Omron CX-Programmer project 新工程 (CX-Programmer 9.42)

# PLC 新PLC1: CP1E N60

## Global symbols (name address type ; comment)
0.04 BOOL  ; 0轴DO2备用
0.06 BOOL  ; 0轴Z相输出
0.07 BOOL  ; 1轴Z相输出
0.10 BOOL  ; 0轴接近零位开关
0.11 BOOL  ; 1轴接近零位开关
100.00 BOOL  ; 0轴脉冲指令
100.01 BOOL  ; 1轴脉冲指令
100.02 BOOL  ; 0轴脉冲方向
100.03 BOOL  ; 1轴脉冲方向
1.04 BOOL  ; 1轴DO2备用
4.10 BOOL  ; 备用
A276 CHANNEL  ; 脉冲输出0的当前值(PV)
A277 CHANNEL  ; 脉冲输出0的当前值(PV)
A278 CHANNEL  ; 脉冲输出1的当前值(PV)
A279 CHANNEL  ; 脉冲输出1的当前值(PV)
A280.00 BOOL  ; 脉冲输出0加速/减速标志
A280.01 BOOL  ; 脉冲输出0上溢/下溢标志
A280.02 BOOL  ; 脉冲输出0输出量设定标志
A280.03 BOOL  ; 脉冲输出0输出完成标志
A280.04 BOOL  ; 脉冲输出0输出中标志
A280.05 BOOL  ; 脉冲输出0无原点标志
A280.06 BOOL  ; 脉冲输出0停止在原点标志
A280.07 BOOL  ; 脉冲输出0输出停止出错标志
A281.00 BOOL  ; 脉冲输出1加速/减速标志
A281.01 BOOL  ; 脉冲输出1上溢/下溢标志
A281.03 BOOL  ; 脉冲输出1输出完成标志
A281.04 BOOL  ; 脉冲输出1输出中标志
A281.05 BOOL  ; 脉冲输出1无原点标志
A281.06 BOOL  ; 脉冲输出1停止在原点标志
A281.07 BOOL  ; 脉冲输出1输出停止出错标志
A444 CHANNEL  ; 脉冲输出0停止出错代码
A445 CHANNEL  ; 脉冲输出1停止出错代码
A540.00 BOOL  ; 脉冲输出0复位位
A540.08 BOOL  ; 脉冲输出0CW限位输入信号标志
A540.09 BOOL  ; 脉冲输出0CCW限位输入信号标志
A540.10 BOOL  ; 脉冲输出0定位完成信号
A541.00 BOOL  ; 脉冲输出1复位位
A541.08 BOOL  ; 脉冲输出1CW限位输入信号标志
A541.09 BOOL  ; 脉冲输出1CCW限位输入信号标志
A541.10 BOOL  ; 脉冲输出1定位完成信号
T201 BOOL  ; 阻挡片气缸1电磁阀
T202 BOOL  ; 阻挡片气缸2电磁阀
T203 BOOL  ; 阻挡片气缸3电磁阀
T204 BOOL  ; 盒子顶出气缸电磁阀
T205 BOOL  ; 机器手气缸1电磁阀
T206 BOOL  ; 机器手气缸2电磁阀
T207 BOOL  ; 旋转90度阻挡气缸1电磁阀
T208 BOOL  ; 旋转90度阻挡气缸2电磁阀
T209 BOOL  ; 上料真空电磁阀
T210 BOOL  ; 下料真空电磁阀
T211 BOOL  ; 吹气电磁阀
T220 BOOL  ; 盒子顶出气缸电磁阀顶出延时
T221 BOOL  ; 盒子顶出气缸电磁阀退回延时
T222 BOOL  ; 光纤物品检测感应2通过延时
T223 BOOL  ; 光纤物品检测感应2顶升延时1
T224 BOOL  ; 机械手1顶出延时1
T225 BOOL  ; 机械手1退回延时1
T226 BOOL  ; 光纤物品检测感应2顶升延时2
T227 BOOL  ; 光纤物品检测感应2顶升延时3
T228 BOOL  ; 开始延时
T229 BOOL  ; 机械手1延时1
T230 BOOL  ; 机械手1延时2
T231 BOOL  ; 机械手1延时3
T232 BOOL  ; 机械手1延时4
T233 BOOL  ; 机械手1延时5
T234 BOOL  ; 机械手1顶出延时2
T235 BOOL  ; 机械手1退回延时2
T236 BOOL  ; 机械手2顶出延时1
T237 BOOL  ; 机械手2退回延时1
T238 BOOL  ; 机械手2顶出延时2
T239 BOOL  ; 机械手2退回延时2
T240 BOOL  ; 机械手2顶出延时3
T241 BOOL  ; 机械手2退回延时3
T242 BOOL  ; 机械手2顶出延时4
T243 BOOL  ; 机械手2退回延时4
T244 BOOL  ; 机械手2顶出延时5
T245 BOOL  ; 机械手2退回延时5
T246 BOOL  ; 机械手2顶出延时6
T247 BOOL  ; 机械手2退回延时6
B_0_ACC_CCW_run 29.05 BOOL  ; 0轴反向运行
B_0_ACC_CW_run 29.03 BOOL  ; 0轴正向运行
B_0_CCW_Interlock 29.08 BOOL  ; 0轴CCW互锁
B_0_CCW_manual 29.14 BOOL  ; 0轴反向手动点动
B_0_CCW_manualing 30.02 BOOL  ; 0轴反向手动点动中
B_0_CW_Interlock 29.07 BOOL  ; 0轴CW互锁
B_0_CW_manual 29.13 BOOL  ; 0轴正向手动点动
B_0_CW_manualing 30.01 BOOL  ; 0轴正向手动点动中
B_0_ORG_POS 31.04 BOOL  ; 0轴原点位置
B_0_ORG_search 30.05 BOOL  ; 0轴原点搜索
B_0_ORG_searched 30.07 BOOL  ; 0轴原点搜索完成
B_0_ORG_searching 30.06 BOOL  ; 0轴原点搜索中
B_0_ORG_seted 30.08 BOOL  ; 0轴原点已定义
B_0_PLS2_CCW_run 28.13 BOOL  ; 0轴反向运行
B_0_PLS2_CW_run 28.11 BOOL  ; 0轴正向运行
B_0_SPED_CCW_run 29.01 BOOL  ; 0轴反向运行
B_0_SPED_CW_run 28.15 BOOL  ; 0轴正向运行
B_0_SRV_ON 31.00 BOOL  ; 0轴伺服ON
B_0_drive_stop 29.11 BOOL  ; 0轴运行停止
B_1_ACC_CCW_run 29.06 BOOL  ; 1轴反向运行
B_1_ACC_CW_run 29.04 BOOL  ; 1轴正向运行
B_1_CCW_Interlock 29.10 BOOL  ; 1轴CCW互锁
B_1_CCW_manual 30.00 BOOL  ; 1轴反向手动点动
B_1_CCW_manualing 30.04 BOOL  ; 1轴反向手动点动中
B_1_CW_Interlock 29.09 BOOL  ; 1轴CW互锁
B_1_CW_manual 29.15 BOOL  ; 1轴正向手动点动
B_1_CW_manualing 30.03 BOOL  ; 1轴正向手动点动中
B_1_ORG_POS 31.05 BOOL  ; 1轴原点位置
B_1_ORG_search 30.09 BOOL  ; 1轴原点搜索
B_1_ORG_searched 30.11 BOOL  ; 1轴原点搜索完成
B_1_ORG_searching 30.10 BOOL  ; 1轴原点搜索中
B_1_ORG_seted 30.12 BOOL  ; 1轴原点已定义
B_1_PLS2_CCW_run 28.14 BOOL  ; 1轴反向运行
B_1_PLS2_CW_run 28.12 BOOL  ; 1轴正向运行
B_1_SPED_CCW_run 29.02 BOOL  ; 1轴反向运行
B_1_SPED_CW_run 29.00 BOOL  ; 1轴正向运行
B_1_SRV_ON 31.01 BOOL  ; 1轴伺服ON
B_1_drive_stop 29.12 BOOL  ; 1轴运行停止
B_LL_1 43.11 BOOL  ; 落料位1
B_LL_2 43.12 BOOL  ; 落料位2
B_LL_3 43.13 BOOL  ; 落料位3
B_LL_4 43.14 BOOL  ; 落料位4
B_POS_DONE 31.03 BOOL  ; 定位结束
B_POS_START_INS 31.02 BOOL  ; 定位开始指令
B_SRV_enabled 30.14 BOOL  ; 伺服自动使能
B_SRV_reset 30.15 BOOL  ; 伺服控制复位
B_SYS_24V_ERR_1 21.04 BOOL  ; 系统24V故障区域1
B_SYS_24V_ERR_2 21.05 BOOL  ; 系统24V故障区域2
B_SYS_24V_ERR_3 21.06 BOOL  ; 系统24V故障区域3
B_SYS_ON_ERR 21.01 BOOL  ; 系统开机故障
B_SYS_RD 20.08 BOOL  ; 系统就绪
B_SYS_airbreaker 20.09 BOOL  ; 系统断路器正常（总）
B_SYS_auto 20.07 BOOL  ; 系统自动（总）
B_SYS_door_ask 20.10 BOOL  ; 系统维修门开门请求（总）
B_SYS_emergency 20.11 BOOL  ; 系统急停（总）
B_SYS_erroring 21.03 BOOL  ; 系统故障中（总）
B_SYS_hold 20.05 BOOL  ; 系统暂停（总）
B_SYS_home 20.12 BOOL  ; 系统工作原点（总）
B_SYS_manual 20.06 BOOL  ; 系统手动（总）
B_SYS_off 20.13 BOOL  ; 系统关机
B_SYS_on 20.14 BOOL  ; 系统开机
B_SYS_oning 20.15 BOOL  ; 系统开机中
B_SYS_reset 20.04 BOOL  ; 系统复位（总）
B_SYS_running 21.00 BOOL  ; 系统运行中
B_SYS_single_cycle 28.10 BOOL  ; 系统单循环（总）
B_SYS_start 20.02 BOOL  ; 系统启动（总）
B_SYS_start_ERR 21.02 BOOL  ; 系统开始故障
B_SYS_stop 20.03 BOOL  ; 系统停止（总）
B_SYS_stoping 20.00 BOOL  ; 系统停止中
B_jog_enabled 30.13 BOOL  ; 手动点动使能
D_0_CCW_acc_Freq 32 DWORD  ; 0轴反向acc目标频率
D_0_CCW_pls2_Freq D1122 DWORD  ; 0轴反向pls2目标频率
D_0_CCW_pls2_PUL D1124 DWORD  ; 0轴反向pls2输出脉冲
D_0_CCW_sped_Freq 38 UDINT  ; 0轴反向点动频率
D_0_CW_acc_Freq 40 DWORD  ; 0轴正向acc目标频率
D_0_CW_pls2_Freq D1102 DWORD  ; 0轴正向pls2目标频率
D_0_CW_pls2_PUL D1104 DWORD  ; 0轴正向pls2输出脉冲
D_0_CW_sped_Freq 46 UDINT  ; 0轴正向点动频率
D_0_user_point_Freq_00 D1000 DWORD  ; 0轴通用位置点频率00
D_0_user_point_Freq_01 D1004 DWORD  ; 0轴通用位置点频率01
D_0_user_point_Freq_02 D1008 DWORD  ; 0轴通用位置点频率02
D_0_user_point_Freq_03 D1012 DWORD  ; 0轴通用位置点频率03
D_0_user_point_Freq_04 D1016 DWORD  ; 0轴通用位置点频率04
D_0_user_point_Freq_05 D1020 DWORD  ; 0轴通用位置点频率05
D_0_user_point_PUL_00 D1002 DWORD  ; 0轴通用位置点脉冲00
D_0_user_point_PUL_01 D1006 DWORD  ; 0轴通用位置点脉冲01
D_0_user_point_PUL_02 D1010 DWORD  ; 0轴通用位置点脉冲02
D_0_user_point_PUL_03 D1014 DWORD  ; 0轴通用位置点脉冲03
D_0_user_point_PUL_04 D1018 DWORD  ; 0轴通用位置点脉冲04
D_0_user_point_PUL_05 D1022 DWORD  ; 0轴通用位置点脉冲05
D_1_CCW_acc_Freq 52 DWORD  ; 1轴反向acc目标频率
D_1_CCW_pls2_Freq D1128 DWORD  ; 1轴反向pls2目标频率
D_1_CCW_pls2_PUL D1130 DWORD  ; 1轴反向pls2输出脉冲
D_1_CCW_sped_Freq 58 UDINT  ; 1轴反向点动频率
D_1_CW_acc_Freq 60 DWORD  ; 1轴正向acc目标频率
D_1_CW_pls2_Freq D1108 DWORD  ; 1轴正向pls2目标频率
D_1_CW_pls2_PUL D1110 DWORD  ; 1轴正向pls2输出脉冲
D_1_CW_sped_Freq 66 UDINT  ; 1轴正向点动频率
D_1_user_point_Freq_00 D1024 DWORD  ; 1轴通用位置点频率00
D_1_user_point_Freq_01 D1028 DWORD  ; 1轴通用位置点频率01
D_1_user_point_Freq_02 D1032 DWORD  ; 1轴通用位置点频率02
D_1_user_point_Freq_03 D1036 DWORD  ; 1轴通用位置点频率03
D_1_user_point_Freq_04 D1040 DWORD  ; 1轴通用位置点频率04
D_1_user_point_Freq_05 D1044 DWORD  ; 1轴通用位置点频率05
D_1_user_point_PUL_00 D1026 DWORD  ; 1轴通用位置点脉冲00
D_1_user_point_PUL_01 D1030 DWORD  ; 1轴通用位置点脉冲01
D_1_user_point_PUL_02 D1034 DWORD  ; 1轴通用位置点脉冲02
D_1_user_point_PUL_03 D1038 DWORD  ; 1轴通用位置点脉冲03
D_1_user_point_PUL_04 D1042 DWORD  ; 1轴通用位置点脉冲04
D_1_user_point_PUL_05 D1046 DWORD  ; 1轴通用位置点脉冲05
END_001_step 22.04 BOOL  ; 结束步01
END_002_step 22.05 BOOL  ; 结束步02
END_FIN_step 22.06 BOOL  ; 结束完成步
HMI_B_0_CCW_manual 132.13 BOOL  ; 0轴反向手动点动
HMI_B_0_CW_manual 132.12 BOOL  ; 0轴正向手动点动
HMI_B_0_ORG_search 132.03 BOOL  ; 0轴原点搜索
HMI_B_0_ORG_seted 132.04 BOOL  ; 0轴原点已定义
HMI_B_0_POS_set 133.02 BOOL  ; 0轴动作点设置
HMI_B_0_PWR_Oning 131.14 BOOL  ; 0轴已上电
HMI_B_0_SRV_ON 132.01 BOOL  ; 0轴伺服ON
HMI_B_0_SRV_Oning 132.00 BOOL  ; 0轴已伺服ON
HMI_B_0_alarm 131.15 BOOL  ; 0轴伺服报警
HMI_B_0_alarm_CLR 132.02 BOOL  ; 0轴警报清除
HMI_B_1_CCW_manual 132.15 BOOL  ; 1轴反向手动点动
HMI_B_1_CW_manual 132.14 BOOL  ; 1轴正向手动点动
HMI_B_1_ORG_search 132.10 BOOL  ; 1轴原点搜索
HMI_B_1_ORG_seted 132.11 BOOL  ; 1轴原点已定义
HMI_B_1_POS_set 133.03 BOOL  ; 1轴动作点设置
HMI_B_1_PWR_Oning 132.05 BOOL  ; 1轴已上电
HMI_B_1_SRV_ON 132.08 BOOL  ; 1轴伺服ON
HMI_B_1_SRV_Oning 132.07 BOOL  ; 1轴已伺服ON
HMI_B_1_alarm 132.06 BOOL  ; 1轴伺服报警
HMI_B_1_alarm_CLR 132.09 BOOL  ; 1轴警报清除
HMI_B_BJ1_QD 130.11 BOOL  ; 步进1启动
HMI_B_BJ1_YG 133.01 BOOL  ; 步进1用光
HMI_B_BJ1_ZQD 133.00 BOOL  ; 步进1再启动
HMI_B_BJ2_QD 130.12 BOOL  ; 步进2启动
HMI_B_BJ3_1 131.00 BOOL  ; 步进3计数器加1
HMI_B_BJ3_1_DONE 131.01 BOOL  ; 步进3计数器结束
HMI_B_BJ3_QD 130.13 BOOL  ; 步进3启动
HMI_B_BJ4_QD 130.14 BOOL  ; 步进4启动
HMI_B_CQF 130.10 BOOL  ; 吹气电磁阀
HMI_B_CQF_ALM 131.13 BOOL  ; 吹气电磁阀报警
HMI_B_DCQGF 130.03 BOOL  ; 盒子顶出气缸电磁阀
HMI_B_DCQGF_ALM 131.06 BOOL  ; 盒子顶出气缸电磁阀报警
HMI_B_PLC_DEBUG 131.02 BOOL  ; PLC单独调试
HMI_B_RBQGF1 130.04 BOOL  ; 机器手气缸1电磁阀
HMI_B_RBQGF1_ALM 131.07 BOOL  ; 机器手气缸1电磁阀报警
HMI_B_RBQGF2 130.05 BOOL  ; 机器手气缸2电磁阀
HMI_B_RBQGF2_ALM 131.08 BOOL  ; 机器手气缸2电磁阀报警
HMI_B_RD_TBC_BT 120.07 BOOL  ; HMI就绪确认
HMI_B_SYS_24V_ERR_1 121.12 BOOL  ; HMI系统24V故障区域1
HMI_B_SYS_24V_ERR_2 121.13 BOOL  ; HMI系统24V故障区域2
HMI_B_SYS_24V_ERR_3 121.14 BOOL  ; HMI系统24V故障区域3
HMI_B_SYS_ON_ERR 121.09 BOOL  ; HMI系统开机故障
HMI_B_SYS_RD 120.15 BOOL  ; HMI系统就绪
HMI_B_SYS_airbreaker 121.01 BOOL  ; HMI系统断路器正常（总）
HMI_B_SYS_auto 120.14 BOOL  ; HMI系统自动（总）
HMI_B_SYS_door_ask 121.02 BOOL  ; HMI系统维修门开门请求（总）
HMI_B_SYS_emergency 121.03 BOOL  ; HMI系统急停（总）
HMI_B_SYS_erroring 121.11 BOOL  ; HMI系统故障中（总）
HMI_B_SYS_hold 120.12 BOOL  ; HMI系统暂停（总）
HMI_B_SYS_home 121.04 BOOL  ; HMI系统工作原点（总）
HMI_B_SYS_manual 120.13 BOOL  ; HMI系统手动（总）
HMI_B_SYS_off 121.05 BOOL  ; HMI系统关机
HMI_B_SYS_on 121.06 BOOL  ; HMI系统开机
HMI_B_SYS_oning 121.07 BOOL  ; HMI系统开机中
HMI_B_SYS_reset 120.11 BOOL  ; HMI系统复位（总）
HMI_B_SYS_running 121.08 BOOL  ; HMI系统运行中
HMI_B_SYS_single_cycle 121.00 BOOL  ; HMI系统单循环（总）
HMI_B_SYS_start 120.09 BOOL  ; HMI系统启动（总）
HMI_B_SYS_start_ERR 121.10 BOOL  ; HMI系统开始故障
HMI_B_SYS_stop 120.10 BOOL  ; HMI系统停止（总）
HMI_B_XZQGF1 130.06 BOOL  ; 旋转90度阻挡气缸1电磁阀
HMI_B_XZQGF1_ALM 131.09 BOOL  ; 旋转90度阻挡气缸1电磁阀报警
HMI_B_XZQGF2 130.07 BOOL  ; 旋转90度阻挡气缸2电磁阀
HMI_B_XZQGF2_ALM 131.10 BOOL  ; 旋转90度阻挡气缸2电磁阀报警
HMI_B_ZDQGF1 130.00 BOOL  ; 阻挡片气缸1电磁阀
HMI_B_ZDQGF1_ALM 131.03 BOOL  ; 阻挡片气缸1电磁阀报警
HMI_B_ZDQGF2 130.01 BOOL  ; 阻挡片气缸2电磁阀
HMI_B_ZDQGF2_ALM 131.04 BOOL  ; 阻挡片气缸2电磁阀报警
HMI_B_ZDQGF3 130.02 BOOL  ; 阻挡片气缸3电磁阀
HMI_B_ZDQGF3_ALM 131.05 BOOL  ; 阻挡片气缸3电磁阀报警
HMI_B_ZKXP1 130.08 BOOL  ; 上料真空电磁阀
HMI_B_ZKXP1_ALM 131.11 BOOL  ; 上料真空电磁阀报警
HMI_B_ZKXP2 130.09 BOOL  ; 下料真空电磁阀
HMI_B_ZKXP2_ALM 131.12 BOOL  ; 下料真空电磁阀报警
HMI_B_auto_BT 120.05 BOOL  ; HMI自动按钮
HMI_B_belt_motor 130.15 BOOL  ; 皮带电机
HMI_B_emergency_BT 120.06 BOOL  ; HMI急停按钮
HMI_B_hold_BT 120.03 BOOL  ; HMI暂停按钮
HMI_B_jog_enabled 132.05 BOOL  ; 手动点动使能
HMI_B_manual_BT 120.04 BOOL  ; HMI手动按钮
HMI_B_reset_BT 120.02 BOOL  ; HMI复位按钮
HMI_B_silence 120.08 BOOL  ; HMI信号灯柱蜂鸣器静音按钮
HMI_B_start_BT 120.00 BOOL  ; HMI开始按钮
HMI_B_stop_BT 120.01 BOOL  ; HMI停止按钮
INIT_001_step 21.11 BOOL  ; 初始步01
INIT_002_step 21.12 BOOL  ; 初始步02
INIT_FIN_step 21.13 BOOL  ; 初始完成步
I_B_0 0.05 BOOL  ; 备用
I_B_0_INP 0.02 BOOL  ; 0轴DO4定位结束
I_B_0_PWR_Oning 0.01 BOOL  ; 0轴DO5已上电
I_B_0_SRV_Oning 0.00 BOOL  ; 0轴DO6外部制动器解除中
I_B_0_alarm 0.03 BOOL  ; 0轴DO3伺服警报
I_B_1 0.08 BOOL  ; 备用
I_B_1_INP 1.02 BOOL  ; 1轴DO4定位结束
I_B_1_PWR_Oning 1.01 BOOL  ; 1轴DO5已上电
I_B_1_SRV_Oning 1.00 BOOL  ; 1轴DO6外部制动器解除中
I_B_1_alarm 1.03 BOOL  ; 1轴DO3伺服警报
I_B_2 0.09 BOOL  ; 备用
I_B_3 1.05 BOOL  ; 备用
I_B_4 1.06 BOOL  ; 备用
I_B_5 1.07 BOOL  ; 备用
I_B_6 1.08 BOOL  ; 备用
I_B_7 1.09 BOOL  ; 备用
I_B_8 1.10 BOOL  ; 备用
I_B_9 1.11 BOOL  ; 备用
I_B_AQSM 3.10 BOOL  ; 安全扫描感应
I_B_BJ1_ALM 5.00 BOOL  ; 步进1报警
I_B_BJ1_POS 5.02 BOOL  ; 步进1到位
I_B_BJ1_RDY 5.01 BOOL  ; 步进1准备
I_B_BJ2_ALM 5.03 BOOL  ; 步进2报警
I_B_BJ2_POS 5.05 BOOL  ; 步进2到位
I_B_BJ2_RDY 5.04 BOOL  ; 步进2准备
I_B_BJ3_1 5.08 BOOL  ; 步进3技术器加1完成
I_B_BJ3_ALM 5.06 BOOL  ; 步进3报警
I_B_BJ3_POS 4.11 BOOL  ; 步进3到位传感器
I_B_BJ3_RDY 5.07 BOOL  ; 步进3准备
I_B_BJ4_ALM 5.09 BOOL  ; 步进4报警
I_B_BJ4_POS 5.11 BOOL  ; 步进4到位
I_B_BJ4_RDY 5.10 BOOL  ; 步进4准备
I_B_DCQG_DOWN 2.07 BOOL  ; 顶出气缸退回
I_B_DCQG_UP 2.06 BOOL  ; 顶出气缸顶出
I_B_GXGY2 3.09 BOOL  ; 光纤物品检测感应2
I_B_GXZQ 3.08 BOOL  ; 光纤抓取高度感应
I_B_JJKG01 3.11 BOOL  ; 接近开关1
I_B_JJKG02 4.00 BOOL  ; 接近开关2
I_B_JJKG03 4.01 BOOL  ; 接近开关3
I_B_JJKG04 4.02 BOOL  ; 接近开关4
I_B_JJKG05 4.03 BOOL  ; 接近开关5
I_B_QYKG1_H 3.04 BOOL  ; 气压开关1高压
I_B_QYKG1_L 3.05 BOOL  ; 气压开关1低压
I_B_QYKG2_H 3.06 BOOL  ; 气压开关2高压
I_B_QYKG2_L 3.07 BOOL  ; 气压开关2低压
I_B_RB10 4.04 BOOL  ; 机器手1原点
I_B_RB1L 4.05 BOOL  ; 机器手1左行程感应
I_B_RB1R 4.06 BOOL  ; 机器手1右行程感应
I_B_RB20 4.07 BOOL  ; 机器手2原点
I_B_RB2L 4.08 BOOL  ; 机器手2左行程感应
I_B_RB2R 4.09 BOOL  ; 机器手2右行程感应
I_B_RBQG1_DOWN 3.01 BOOL  ; 机械手1顶出
I_B_RBQG1_UP 3.00 BOOL  ; 机械手1退回
I_B_RBQG2_DOWN 3.03 BOOL  ; 机械手2顶出
I_B_RBQG2_UP 3.02 BOOL  ; 机械手2退回
I_B_XZQG1_DOWN 2.09 BOOL  ; 旋转1退回
I_B_XZQG1_UP 2.08 BOOL  ; 旋转1顶出
I_B_XZQG2_DOWN 2.11 BOOL  ; 旋转2退回
I_B_XZQG2_UP 2.10 BOOL  ; 旋转2顶出
I_B_ZDQG1_DOWN 2.01 BOOL  ; 阻挡气缸1退回
I_B_ZDQG1_UP 2.00 BOOL  ; 阻挡气缸1顶出
I_B_ZDQG2_DOWN 2.03 BOOL  ; 阻挡气缸2退回
I_B_ZDQG2_UP 2.02 BOOL  ; 阻挡气缸2顶出
I_B_ZDQG3_DOWN 2.05 BOOL  ; 阻挡气缸3退回
I_B_ZDQG3_UP 2.04 BOOL  ; 阻挡气缸3顶出
PLC11_001_step 22.07 BOOL  ; PLC11步001
PLC11_002_step 22.08 BOOL  ; PLC11步002
PLC11_003_step 22.09 BOOL  ; PLC11步003
PLC11_004_step 22.10 BOOL  ; PLC11步004
PLC11_005_step 22.11 BOOL  ; PLC11步005
PLC11_006_step 22.12 BOOL  ; PLC11步006
PLC11_007_step 22.13 BOOL  ; PLC11步007
PLC11_008_step 22.14 BOOL  ; PLC11步008
PLC11_009_step 22.15 BOOL  ; PLC11步009
PLC11_010_step 23.00 BOOL  ; PLC11步010
PLC11_011_step 23.01 BOOL  ; PLC11步011
PLC11_012_step 23.02 BOOL  ; PLC11步012
PLC11_013_step 23.03 BOOL  ; PLC11步013
PLC11_014_step 23.04 BOOL  ; PLC11步014
PLC11_015_step 23.05 BOOL  ; PLC11步015
PLC11_016_step 23.06 BOOL  ; PLC11步016
PLC11_017_step 23.07 BOOL  ; PLC11步017
PLC11_018_step 23.08 BOOL  ; PLC11步018
PLC11_019_step 23.09 BOOL  ; PLC11步019
PLC11_020_step 23.10 BOOL  ; PLC11步020
PLC11_021_step 23.11 BOOL  ; PLC11步021
PLC11_022_step 23.12 BOOL  ; PLC11步022
PLC11_023_step 23.13 BOOL  ; PLC11步023
PLC11_024_step 23.14 BOOL  ; PLC11步024
PLC11_025_step 23.15 BOOL  ; PLC11步025
PLC11_026_step 24.00 BOOL  ; PLC11步026
PLC11_027_step 24.01 BOOL  ; PLC11步027
PLC11_028_step 24.02 BOOL  ; PLC11步028
PLC11_029_step 24.03 BOOL  ; PLC11步029
PLC11_030_step 24.04 BOOL  ; PLC11步030
PLC11_031_step 24.05 BOOL  ; PLC11步031
PLC11_032_step 24.06 BOOL  ; PLC11步032
PLC11_033_step 24.07 BOOL  ; PLC11步033
PLC11_034_step 24.08 BOOL  ; PLC11步034
PLC11_035_step 24.09 BOOL  ; PLC11步035
PLC11_036_step 24.10 BOOL  ; PLC11步036
PLC11_037_step 24.11 BOOL  ; PLC11步037
PLC11_038_step 24.12 BOOL  ; PLC11步038
PLC11_039_step 24.13 BOOL  ; PLC11步039
PLC11_040_step 24.14 BOOL  ; PLC11步040
PLC11_041_step 24.15 BOOL  ; PLC11步041
PLC11_042_step 25.00 BOOL  ; PLC11步042
PLC11_043_step 25.01 BOOL  ; PLC11步043
PLC11_044_step 25.02 BOOL  ; PLC11步044
PLC11_045_step 25.03 BOOL  ; PLC11步045
PLC11_046_step 25.04 BOOL  ; PLC11步046
PLC11_047_step 25.05 BOOL  ; PLC11步047
PLC11_048_step 25.06 BOOL  ; PLC11步048
PLC11_049_step 25.07 BOOL  ; PLC11步049
PLC11_050_step 25.08 BOOL  ; PLC11步050
PLC11_051_step 25.09 BOOL  ; PLC11步051
PLC11_052_step 25.10 BOOL  ; PLC11步052
PLC11_053_step 25.11 BOOL  ; PLC11步053
PLC11_054_step 25.12 BOOL  ; PLC11步054
PLC11_055_step 25.13 BOOL  ; PLC11步055
PLC11_056_step 25.14 BOOL  ; PLC11步056
PLC11_057_step 25.15 BOOL  ; PLC11步057
PLC11_058_step 26.00 BOOL  ; PLC11步058
PLC11_059_step 26.01 BOOL  ; PLC11步059
PLC11_060_step 26.02 BOOL  ; PLC11步060
PLC11_061_step 26.03 BOOL  ; PLC11步061
PLC11_062_step 26.04 BOOL  ; PLC11步062
PLC11_063_step 26.05 BOOL  ; PLC11步063
PLC11_064_step 26.06 BOOL  ; PLC11步064
PLC11_065_step 26.07 BOOL  ; PLC11步065
PLC11_066_step 26.08 BOOL  ; PLC11步066
PLC11_067_step 26.09 BOOL  ; PLC11步067
PLC11_068_step 26.10 BOOL  ; PLC11步068
PLC11_069_step 26.11 BOOL  ; PLC11步069
PLC11_070_step 26.12 BOOL  ; PLC11步070
PLC11_071_step 26.13 BOOL  ; PLC11步071
PLC11_072_step 26.14 BOOL  ; PLC11步072
PLC11_073_step 26.15 BOOL  ; PLC11步073
PLC11_074_step 27.00 BOOL  ; PLC11步074
PLC11_075_step 27.01 BOOL  ; PLC11步075
PLC11_076_step 27.02 BOOL  ; PLC11步076
PLC11_077_step 27.03 BOOL  ; PLC11步077
PLC11_078_step 27.04 BOOL  ; PLC11步078
PLC11_079_step 27.05 BOOL  ; PLC11步079
PLC11_080_step 27.06 BOOL  ; PLC11步080
PLC11_081_step 27.07 BOOL  ; PLC11步081
PLC11_082_step 27.08 BOOL  ; PLC11步082
PLC11_083_step 27.09 BOOL  ; PLC11步083
PLC11_084_step 27.10 BOOL  ; PLC11步084
PLC11_085_step 27.11 BOOL  ; PLC11步085
PLC11_086_step 27.12 BOOL  ; PLC11步086
PLC11_087_step 27.13 BOOL  ; PLC11步087
PLC11_088_step 27.14 BOOL  ; PLC11步088
PLC11_089_step 27.15 BOOL  ; PLC11步089
PLC11_090_step 28.00 BOOL  ; PLC11步090
PLC11_091_step 28.01 BOOL  ; PLC11步091
PLC11_092_step 28.02 BOOL  ; PLC11步092
PLC11_093_step 28.03 BOOL  ; PLC11步093
PLC11_094_step 28.04 BOOL  ; PLC11步094
PLC11_095_step 28.05 BOOL  ; PLC11步095
PLC11_096_step 28.06 BOOL  ; PLC11步096
PLC11_097_step 28.07 BOOL  ; PLC11步097
PLC11_098_step 28.08 BOOL  ; PLC11步098
PLC11_099_step 28.09 BOOL  ; PLC11步099
PLC11_100_step 31.06 BOOL  ; PLC11步100
PLC11_101_step 31.07 BOOL  ; PLC11步101
PLC11_102_step 31.08 BOOL  ; PLC11步102
PLC11_103_step 31.09 BOOL  ; PLC11步103
PLC11_104_step 31.10 BOOL  ; PLC11步104
PLC11_105_step 31.11 BOOL  ; PLC11步105
PLC11_106_step 31.12 BOOL  ; PLC11步106
PLC11_107_step 31.13 BOOL  ; PLC11步107
PLC11_108_step 31.14 BOOL  ; PLC11步108
PLC11_109_step 31.15 BOOL  ; PLC11步109
PLC11_110_step 34.00 BOOL  ; PLC11步110
PLC11_111_step 34.01 BOOL  ; PLC11步111
PLC11_112_step 34.02 BOOL  ; PLC11步112
PLC11_113_step 34.03 BOOL  ; PLC11步113
PLC11_114_step 34.04 BOOL  ; PLC11步114
PLC11_115_step 34.05 BOOL  ; PLC11步115
PLC11_116_step 34.06 BOOL  ; PLC11步116
PLC11_117_step 34.07 BOOL  ; PLC11步117
PLC11_118_step 34.08 BOOL  ; PLC11步118
PLC11_119_step 34.09 BOOL  ; PLC11步119
PLC11_120_step 34.10 BOOL  ; PLC11步120
PLC11_121_step 34.11 BOOL  ; PLC11步121
PLC11_122_step 34.12 BOOL  ; PLC11步122
PLC11_123_step 34.13 BOOL  ; PLC11步123
PLC11_124_step 34.14 BOOL  ; PLC11步124
PLC11_125_step 34.15 BOOL  ; PLC11步125
PLC11_126_step 35.00 BOOL  ; PLC11步126
PLC11_127_step 35.01 BOOL  ; PLC11步127
PLC11_128_step 35.02 BOOL  ; PLC11步128
PLC11_129_step 35.03 BOOL  ; PLC11步129
PLC11_130_step 35.04 BOOL  ; PLC11步130
PLC11_131_step 35.05 BOOL  ; PLC11步131
PLC11_132_step 35.06 BOOL  ; PLC11步132
PLC11_133_step 35.07 BOOL  ; PLC11步133
PLC11_134_step 35.08 BOOL  ; PLC11步134
PLC11_135_step 35.09 BOOL  ; PLC11步135
PLC11_136_step 35.10 BOOL  ; PLC11步136
PLC11_137_step 35.11 BOOL  ; PLC11步137
PLC11_138_step 35.12 BOOL  ; PLC11步138
PLC11_139_step 35.13 BOOL  ; PLC11步139
PLC11_140_step 35.14 BOOL  ; PLC11步140
PLC11_141_step 35.15 BOOL  ; PLC11步141
PLC11_142_step 36.00 BOOL  ; PLC11步142
PLC11_143_step 36.01 BOOL  ; PLC11步143
PLC11_144_step 36.02 BOOL  ; PLC11步144
PLC11_145_step 36.03 BOOL  ; PLC11步145
PLC11_146_step 36.04 BOOL  ; PLC11步146
PLC11_147_step 36.05 BOOL  ; PLC11步147
PLC11_148_step 36.06 BOOL  ; PLC11步148
PLC11_149_step 36.07 BOOL  ; PLC11步149
PLC11_150_step 36.08 BOOL  ; PLC11步150
PLC11_151_step 36.09 BOOL  ; PLC11步151
PLC11_152_step 36.10 BOOL  ; PLC11步152
PLC11_153_step 36.11 BOOL  ; PLC11步153
PLC11_154_step 36.12 BOOL  ; PLC11步154
PLC11_155_step 36.13 BOOL  ; PLC11步155
PLC11_156_step 36.14 BOOL  ; PLC11步156
PLC11_157_step 36.15 BOOL  ; PLC11步157
PLC11_158_step 37.00 BOOL  ; PLC11步158
PLC11_159_step 37.01 BOOL  ; PLC11步159
PLC11_160_step 37.02 BOOL  ; PLC11步160
PLC11_161_step 37.03 BOOL  ; PLC11步161
PLC11_162_step 37.04 BOOL  ; PLC11步162
PLC11_163_step 37.05 BOOL  ; PLC11步163
PLC11_164_step 37.06 BOOL  ; PLC11步164
PLC11_165_step 37.07 BOOL  ; PLC11步165
PLC11_166_step 37.08 BOOL  ; PLC11步166
PLC11_167_step 37.09 BOOL  ; PLC11步167
PLC11_168_step 37.10 BOOL  ; PLC11步168
PLC11_169_step 37.11 BOOL  ; PLC11步169
PLC11_170_step 37.12 BOOL  ; PLC11步170
PLC11_171_step 37.13 BOOL  ; PLC11步171
PLC11_172_step 37.14 BOOL  ; PLC11步172
PLC11_173_step 37.15 BOOL  ; PLC11步173
PLC11_174_step 42.00 BOOL  ; PLC11步174
PLC11_175_step 42.01 BOOL  ; PLC11步175
PLC11_176_step 42.02 BOOL  ; PLC11步176
PLC11_177_step 42.03 BOOL  ; PLC11步177
PLC11_178_step 42.04 BOOL  ; PLC11步178
PLC11_179_step 42.05 BOOL  ; PLC11步179
PLC11_180_step 42.06 BOOL  ; PLC11步180
PLC11_181_step 42.07 BOOL  ; PLC11步181
PLC11_182_step 42.08 BOOL  ; PLC11步182
PLC11_183_step 42.09 BOOL  ; PLC11步183
PLC11_184_step 42.10 BOOL  ; PLC11步184
PLC11_185_step 42.11 BOOL  ; PLC11步185
PLC11_186_step 42.12 BOOL  ; PLC11步186
PLC11_187_step 42.13 BOOL  ; PLC11步187
PLC11_188_step 42.14 BOOL  ; PLC11步188
PLC11_189_step 42.15 BOOL  ; PLC11步189
PLC11_190_step 43.00 BOOL  ; PLC11步190
PLC11_191_step 43.01 BOOL  ; PLC11步191
PLC11_192_step 43.02 BOOL  ; PLC11步192
PLC11_193_step 43.03 BOOL  ; PLC11步193
PLC11_194_step 43.04 BOOL  ; PLC11步194
PLC11_195_step 43.05 BOOL  ; PLC11步195
PLC11_196_step 43.06 BOOL  ; PLC11步196
PLC11_197_step 43.07 BOOL  ; PLC11步197
PLC11_198_step 43.08 BOOL  ; PLC11步198
PLC11_199_step 43.09 BOOL  ; PLC11步199
PLC11_200_step 43.10 BOOL  ; PLC11步200
PLC11_END_step 21.10 BOOL  ; PLC结束步
PLC11_INIT_step 21.07 BOOL  ; PLC初始步
PLC11_start_step 21.08 BOOL  ; PLC开始步
PLC11_stop_step 21.09 BOOL  ; PLC停止步
Q_B_0_CL 100.04 BOOL  ; 0轴DI2错误计数器复位
Q_B_0_GAIN 101.05 BOOL  ; 0轴DI9增益转换
Q_B_0_NOT 101.03 BOOL  ; 0轴DI6负方向驱动禁止
Q_B_0_POT 101.04 BOOL  ; 0轴DI7正方向驱动禁止
Q_B_0_SRV_ON 101.06 BOOL  ; 0轴DI1伺服ON
Q_B_0_alarm_CLR 101.07 BOOL  ; 0轴DI5警报清除
Q_B_1 6.00 BOOL  ; 备用
Q_B_10 6.09 BOOL  ; 备用
Q_B_11 6.10 BOOL  ; 备用
Q_B_12 6.11 BOOL  ; 备用
Q_B_14 101.01 BOOL  ; 备用
Q_B_15 101.02 BOOL  ; 备用
Q_B_16 102.00 BOOL  ; 备用
Q_B_17 102.01 BOOL  ; 备用
Q_B_18 102.02 BOOL  ; 备用
Q_B_1_CL 100.05 BOOL  ; 1轴DI2错误计数器复位
Q_B_1_GAIN 102.05 BOOL  ; 1轴DI9增益转换
Q_B_1_NOT 102.03 BOOL  ; 1轴DI6负方向驱动禁止
Q_B_1_POT 102.04 BOOL  ; 1轴DI7正方向驱动禁止
Q_B_1_SRV_ON 102.06 BOOL  ; 1轴DI1伺服ON
Q_B_1_alarm_CLR 102.07 BOOL  ; 1轴DI5警报清除
Q_B_2 6.01 BOOL  ; 备用
Q_B_3 6.02 BOOL  ; 备用
Q_B_4 6.03 BOOL  ; 备用
Q_B_5 6.04 BOOL  ; 备用
Q_B_6 6.05 BOOL  ; 备用
Q_B_7 6.06 BOOL  ; 备用
Q_B_8 6.07 BOOL  ; 备用
Q_B_9 6.08 BOOL  ; 备用
Q_B_BJ1_QD 106.00 BOOL  ; 步进1启动
Q_B_BJ1_YG 106.07 BOOL  ; 步进1用光
Q_B_BJ1_ZQD 106.06 BOOL  ; 步进1再启动
Q_B_BJ2_QD 106.01 BOOL  ; 步进2启动
Q_B_BJ3_1 106.03 BOOL  ; 步进3计数器加1
Q_B_BJ3_1_DONE 106.04 BOOL  ; 步进3计数器结束
Q_B_BJ3_QD 106.02 BOOL  ; 步进3启动
Q_B_BJ4_QD 106.05 BOOL  ; 步进4启动
Q_B_CQF 104.02 BOOL  ; 吹气电磁阀
Q_B_DCQGF 103.03 BOOL  ; 盒子顶出气缸电磁阀
Q_B_GY 105.07 BOOL  ; 标准光源（继电器）
Q_B_HZM_ALM 105.00 BOOL  ; 盒子满蜂鸣器
Q_B_HZM_RED 104.07 BOOL  ; 盒子满红灯
Q_B_LIGHT_ALM 104.06 BOOL  ; 三色灯自带故障蜂鸣器
Q_B_LIGHT_GREEN 104.05 BOOL  ; 三色顶部指示灯绿
Q_B_LIGHT_RED 104.03 BOOL  ; 三色顶部指示灯红
Q_B_LIGHT_YELLOW 104.04 BOOL  ; 三色顶部指示灯黄
Q_B_PULS 105.01 BOOL  ; 总计数器
Q_B_PULS_1 105.02 BOOL  ; 分计数器1
Q_B_PULS_2 105.03 BOOL  ; 分计数器2
Q_B_PULS_3 105.04 BOOL  ; 分计数器3
Q_B_PULS_4 105.05 BOOL  ; 分计数器4
Q_B_PULS_5 105.06 BOOL  ; 分计数器5
Q_B_RBQGF1 103.04 BOOL  ; 机器手气缸1电磁阀
Q_B_RBQGF2 103.05 BOOL  ; 机器手气缸2电磁阀
Q_B_SSR_1 100.06 BOOL  ; SSR固态继电器1
Q_B_SSR_2 100.07 BOOL  ; SSR固态继电器2
Q_B_XZQGF1 103.06 BOOL  ; 旋转90度阻挡气缸1电磁阀
Q_B_XZQGF2 103.07 BOOL  ; 旋转90度阻挡气缸2电磁阀
Q_B_ZDQGF1 103.00 BOOL  ; 阻挡片气缸1电磁阀
Q_B_ZDQGF2 103.01 BOOL  ; 阻挡片气缸2电磁阀
Q_B_ZDQGF3 103.02 BOOL  ; 阻挡片气缸3电磁阀
Q_B_ZKXP1 104.00 BOOL  ; 上料真空电磁阀
Q_B_ZKXP2 104.01 BOOL  ; 下料真空电磁阀
Q_B_belt_motor 101.00 BOOL  ; 皮带电机
W_0_CCW_acc_ACCDEC 72 CHANNEL  ; 0轴反向acc加减速率
W_0_CCW_pls2_ACC D1120 CHANNEL  ; 0轴反向pls2加速率
W_0_CCW_pls2_DEC D1121 CHANNEL  ; 0轴反向pls2减速率
W_0_CW_acc_ACCDEC 75 CHANNEL  ; 0轴正向acc加减速率
W_0_CW_pls2_ACC D1100 CHANNEL  ; 0轴正向pls2加速率
W_0_CW_pls2_DEC D1101 CHANNEL  ; 0轴正向pls2减速率
W_1_CCW_acc_ACCDEC 78 CHANNEL  ; 1轴反向acc加减速率
W_1_CCW_pls2_ACC D1126 CHANNEL  ; 1轴反向pls2加速率
W_1_CCW_pls2_DEC D1127 CHANNEL  ; 1轴反向pls2减速率
W_1_CW_acc_ACCDEC 81 CHANNEL  ; 1轴正向acc加减速率
W_1_CW_pls2_ACC D1106 CHANNEL  ; 1轴正向pls2加速率
W_1_CW_pls2_DEC D1107 CHANNEL  ; 1轴正向pls2减速率
W_axis_selection 20.01 BOOL  ; 选择0-0轴，1-1轴
start_001_step 21.14 BOOL  ; 开始步01
start_002_step 21.15 BOOL  ; 开始步02
start_FIN_step 22.00 BOOL  ; 开始完成步
stop_001_step 22.01 BOOL  ; 停止步01
stop_002_step 22.02 BOOL  ; 停止步02
stop_FIN_step 22.03 BOOL  ; 停止完成步

## Program 新程序1 (cyclic task 0)

### Section _1601_MODE

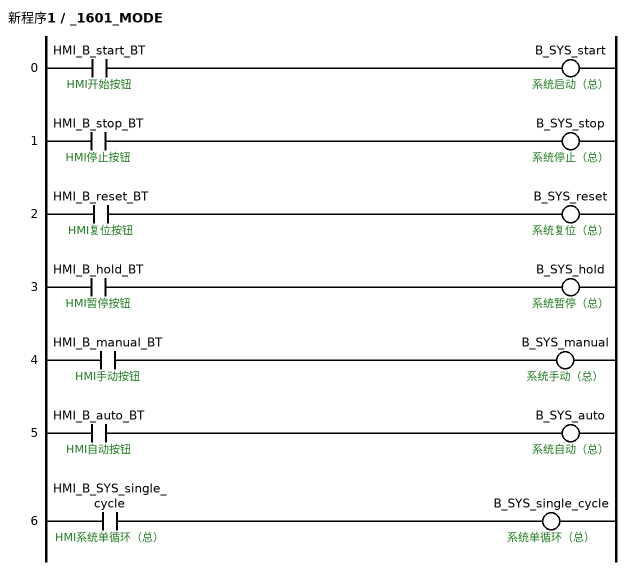
; rung 0
LD HMI_B_start_BT  ; HMI开始按钮
OUT B_SYS_start  ; 系统启动（总）
; rung 1
LD HMI_B_stop_BT  ; HMI停止按钮
OUT B_SYS_stop  ; 系统停止（总）
; rung 2
LD HMI_B_reset_BT  ; HMI复位按钮
OUT B_SYS_reset  ; 系统复位（总）
; rung 3
LD HMI_B_hold_BT  ; HMI暂停按钮
OUT B_SYS_hold  ; 系统暂停（总）
; rung 4
LD HMI_B_manual_BT  ; HMI手动按钮
OUT B_SYS_manual  ; 系统手动（总）
; rung 5
LD HMI_B_auto_BT  ; HMI自动按钮
OUT B_SYS_auto  ; 系统自动（总）
; rung 6
LD HMI_B_SYS_single_cycle  ; HMI系统单循环（总）
OUT B_SYS_single_cycle  ; 系统单循环（总）

### Section _1601_CONDITION

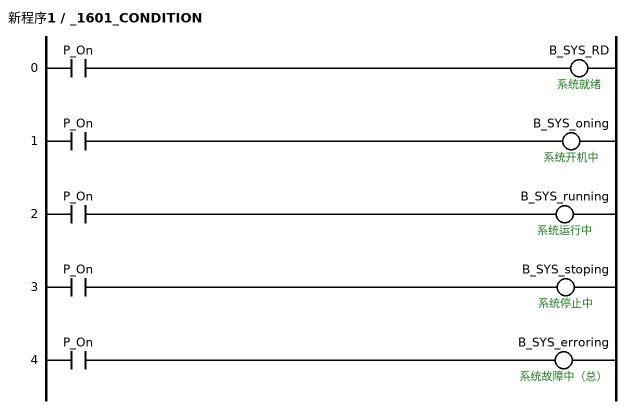
; rung 0
LD P_On
OUT B_SYS_RD  ; 系统就绪
; rung 1
LD P_On
OUT B_SYS_oning  ; 系统开机中
; rung 2
LD P_On
OUT B_SYS_running  ; 系统运行中
; rung 3
LD P_On
OUT B_SYS_stoping  ; 系统停止中
; rung 4
LD P_On
OUT B_SYS_erroring  ; 系统故障中（总）

### Section _1601_HMI

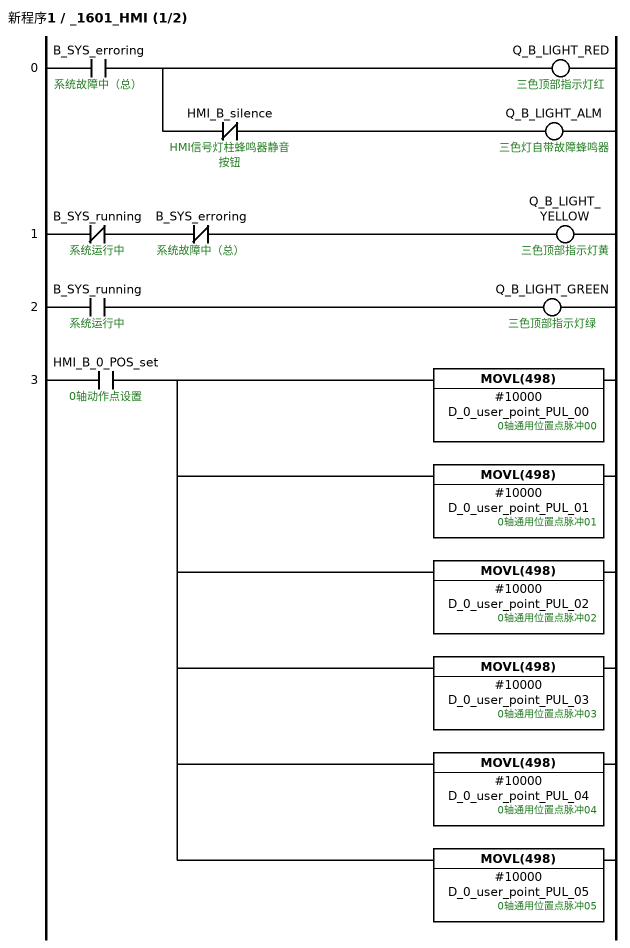
; rung 0
LD B_SYS_erroring  ; 系统故障中（总）
OUT Q_B_LIGHT_RED  ; 三色顶部指示灯红
ANDNOT HMI_B_silence  ; HMI信号灯柱蜂鸣器静音按钮
OUT Q_B_LIGHT_ALM  ; 三色灯自带故障蜂鸣器
; rung 1
LDNOT B_SYS_running  ; 系统运行中
ANDNOT B_SYS_erroring  ; 系统故障中（总）
OUT Q_B_LIGHT_YELLOW  ; 三色顶部指示灯黄
; rung 2
LD B_SYS_running  ; 系统运行中
OUT Q_B_LIGHT_GREEN  ; 三色顶部指示灯绿
; rung 3
LD HMI_B_0_POS_set  ; 0轴动作点设置
MOVL(498) #10000 D_0_user_point_PUL_00  ; 0轴通用位置点脉冲00
MOVL(498) #10000 D_0_user_point_PUL_01  ; 0轴通用位置点脉冲01
MOVL(498) #10000 D_0_user_point_PUL_02  ; 0轴通用位置点脉冲02
MOVL(498) #10000 D_0_user_point_PUL_03  ; 0轴通用位置点脉冲03
MOVL(498) #10000 D_0_user_point_PUL_04  ; 0轴通用位置点脉冲04
MOVL(498) #10000 D_0_user_point_PUL_05  ; 0轴通用位置点脉冲05

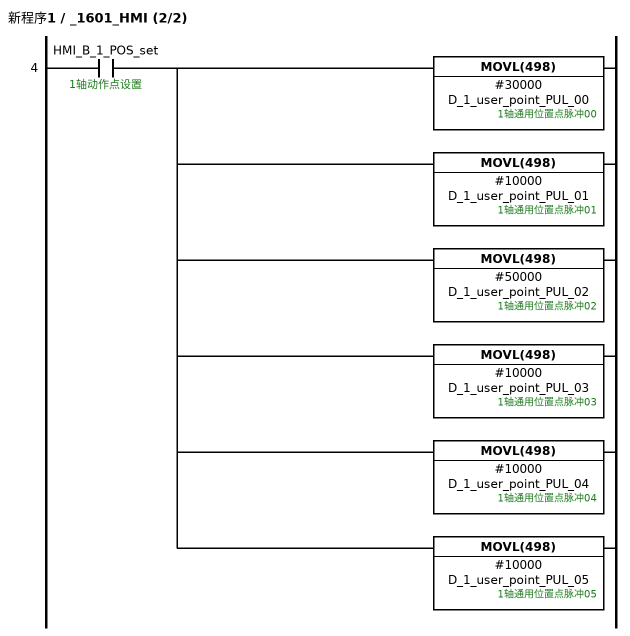
; rung 4
LD HMI_B_1_POS_set  ; 1轴动作点设置
MOVL(498) #30000 D_1_user_point_PUL_00  ; 1轴通用位置点脉冲00
MOVL(498) #10000 D_1_user_point_PUL_01  ; 1轴通用位置点脉冲01
MOVL(498) #50000 D_1_user_point_PUL_02  ; 1轴通用位置点脉冲02
MOVL(498) #10000 D_1_user_point_PUL_03  ; 1轴通用位置点脉冲03
MOVL(498) #10000 D_1_user_point_PUL_04  ; 1轴通用位置点脉冲04
MOVL(498) #10000 D_1_user_point_PUL_05  ; 1轴通用位置点脉冲05

### Section _1601_OUT

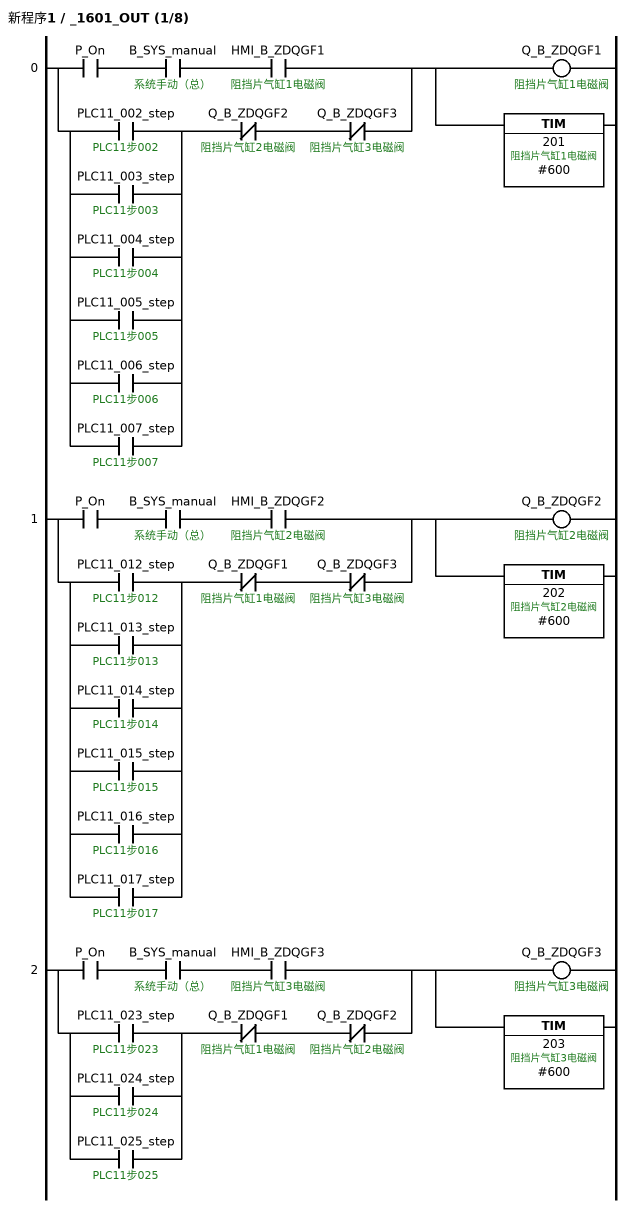
; rung 0
LD P_On
AND B_SYS_manual  ; 系统手动（总）
AND HMI_B_ZDQGF1  ; 阻挡片气缸1电磁阀
LD PLC11_002_step  ; PLC11步002
OR PLC11_003_step  ; PLC11步003
OR PLC11_004_step  ; PLC11步004
OR PLC11_005_step  ; PLC11步005
OR PLC11_006_step  ; PLC11步006
OR PLC11_007_step  ; PLC11步007
ANDNOT Q_B_ZDQGF2  ; 阻挡片气缸2电磁阀
ANDNOT Q_B_ZDQGF3  ; 阻挡片气缸3电磁阀
ORLD
OUT Q_B_ZDQGF1  ; 阻挡片气缸1电磁阀
TIM 201 #600  ; 阻挡片气缸1电磁阀
; rung 1
LD P_On
AND B_SYS_manual  ; 系统手动（总）
AND HMI_B_ZDQGF2  ; 阻挡片气缸2电磁阀
LD PLC11_012_step  ; PLC11步012
OR PLC11_013_step  ; PLC11步013
OR PLC11_014_step  ; PLC11步014
OR PLC11_015_step  ; PLC11步015
OR PLC11_016_step  ; PLC11步016
OR PLC11_017_step  ; PLC11步017
ANDNOT Q_B_ZDQGF1  ; 阻挡片气缸1电磁阀
ANDNOT Q_B_ZDQGF3  ; 阻挡片气缸3电磁阀
ORLD
OUT Q_B_ZDQGF2  ; 阻挡片气缸2电磁阀
TIM 202 #600  ; 阻挡片气缸2电磁阀
; rung 2
LD P_On
AND B_SYS_manual  ; 系统手动（总）
AND HMI_B_ZDQGF3  ; 阻挡片气缸3电磁阀
LD PLC11_023_step  ; PLC11步023
OR PLC11_024_step  ; PLC11步024
OR PLC11_025_step  ; PLC11步025
ANDNOT Q_B_ZDQGF1  ; 阻挡片气缸1电磁阀
ANDNOT Q_B_ZDQGF2  ; 阻挡片气缸2电磁阀
ORLD
OUT Q_B_ZDQGF3  ; 阻挡片气缸3电磁阀
TIM 203 #600  ; 阻挡片气缸3电磁阀

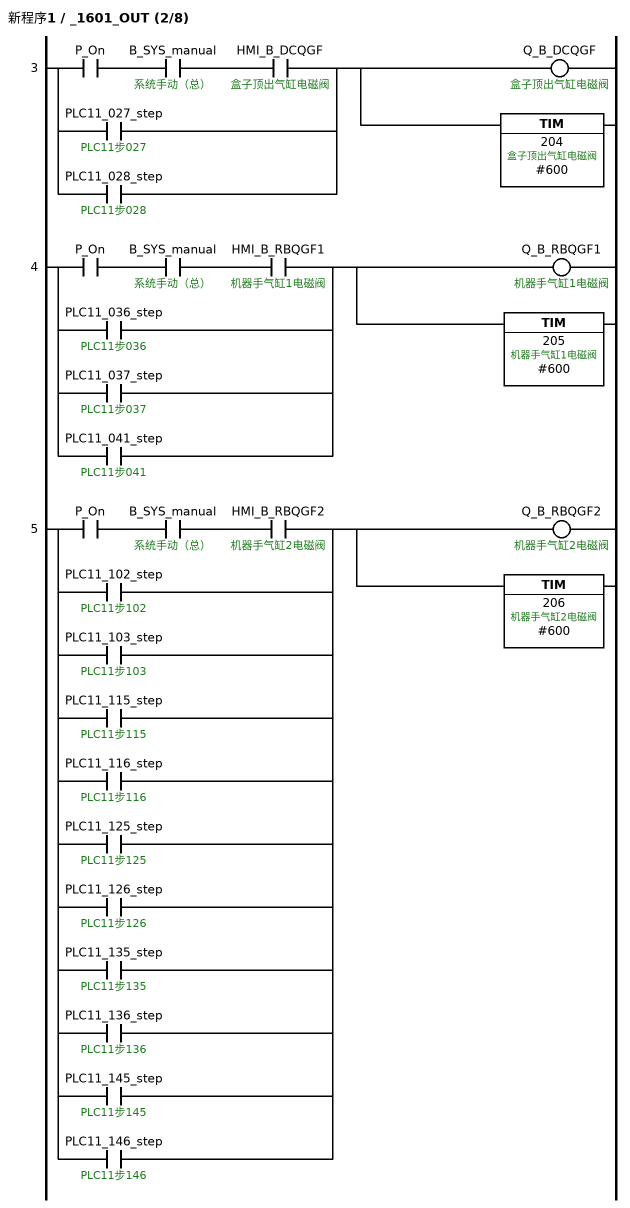
; rung 3
LD P_On
AND B_SYS_manual  ; 系统手动（总）
AND HMI_B_DCQGF  ; 盒子顶出气缸电磁阀
OR PLC11_027_step  ; PLC11步027
OR PLC11_028_step  ; PLC11步028
OUT Q_B_DCQGF  ; 盒子顶出气缸电磁阀
TIM 204 #600  ; 盒子顶出气缸电磁阀
; rung 4
LD P_On
AND B_SYS_manual  ; 系统手动（总）
AND HMI_B_RBQGF1  ; 机器手气缸1电磁阀
OR PLC11_036_step  ; PLC11步036
OR PLC11_037_step  ; PLC11步037
OR PLC11_041_step  ; PLC11步041
OUT Q_B_RBQGF1  ; 机器手气缸1电磁阀
TIM 205 #600  ; 机器手气缸1电磁阀
; rung 5
LD P_On
AND B_SYS_manual  ; 系统手动（总）
AND HMI_B_RBQGF2  ; 机器手气缸2电磁阀
OR PLC11_102_step  ; PLC11步102
OR PLC11_103_step  ; PLC11步103
LD PLC11_115_step  ; PLC11步115
OR PLC11_116_step  ; PLC11步116
ORLD
LD PLC11_125_step  ; PLC11步125
OR PLC11_126_step  ; PLC11步126
ORLD
LD PLC11_135_step  ; PLC11步135
OR PLC11_136_step  ; PLC11步136
ORLD
LD PLC11_145_step  ; PLC11步145
OR PLC11_146_step  ; PLC11步146
ORLD
OUT Q_B_RBQGF2  ; 机器手气缸2电磁阀
TIM 206 #600  ; 机器手气缸2电磁阀

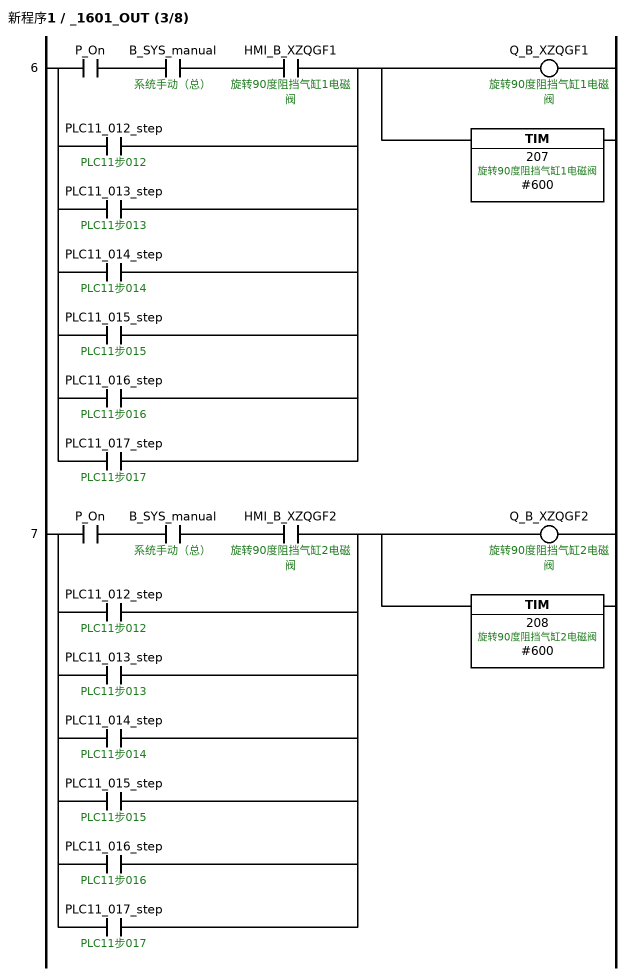
; rung 6
LD P_On
AND B_SYS_manual  ; 系统手动（总）
AND HMI_B_XZQGF1  ; 旋转90度阻挡气缸1电磁阀
OR PLC11_012_step  ; PLC11步012
OR PLC11_013_step  ; PLC11步013
OR PLC11_014_step  ; PLC11步014
OR PLC11_015_step  ; PLC11步015
OR PLC11_016_step  ; PLC11步016
OR PLC11_017_step  ; PLC11步017
OUT Q_B_XZQGF1  ; 旋转90度阻挡气缸1电磁阀
TIM 207 #600  ; 旋转90度阻挡气缸1电磁阀
; rung 7
LD P_On
AND B_SYS_manual  ; 系统手动（总）
AND HMI_B_XZQGF2  ; 旋转90度阻挡气缸2电磁阀
OR PLC11_012_step  ; PLC11步012
OR PLC11_013_step  ; PLC11步013
OR PLC11_014_step  ; PLC11步014
OR PLC11_015_step  ; PLC11步015
OR PLC11_016_step  ; PLC11步016
OR PLC11_017_step  ; PLC11步017
OUT Q_B_XZQGF2  ; 旋转90度阻挡气缸2电磁阀
TIM 208 #600  ; 旋转90度阻挡气缸2电磁阀

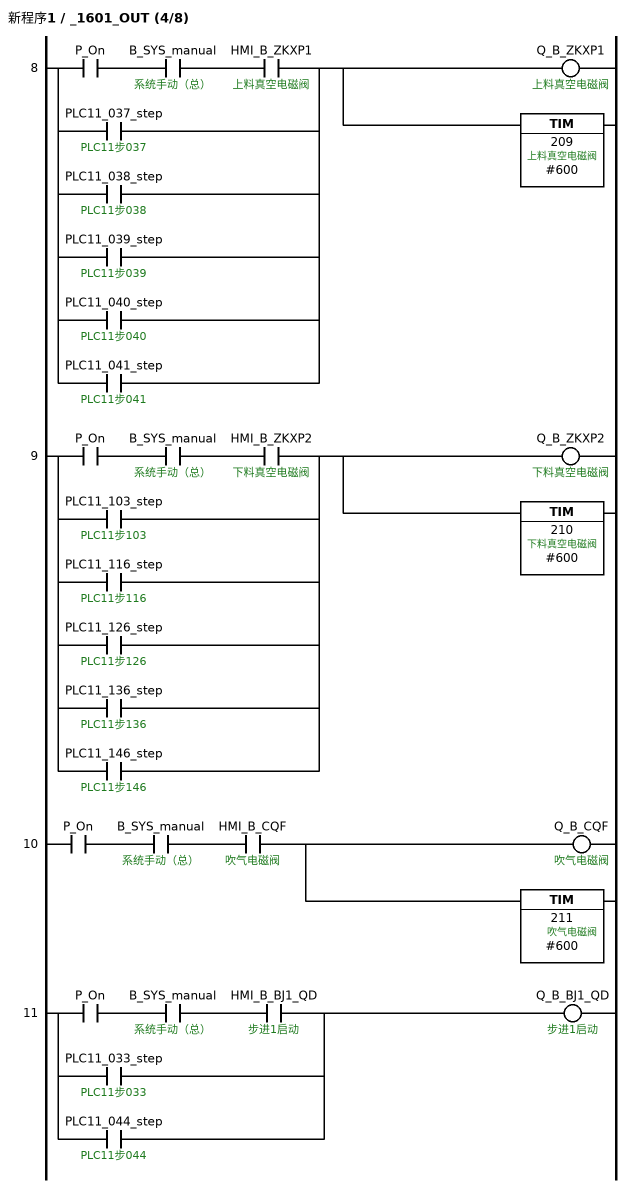
; rung 8
LD P_On
AND B_SYS_manual  ; 系统手动（总）
AND HMI_B_ZKXP1  ; 上料真空电磁阀
OR PLC11_037_step  ; PLC11步037
OR PLC11_038_step  ; PLC11步038
OR PLC11_039_step  ; PLC11步039
OR PLC11_040_step  ; PLC11步040
OR PLC11_041_step  ; PLC11步041
OUT Q_B_ZKXP1  ; 上料真空电磁阀
TIM 209 #600  ; 上料真空电磁阀
; rung 9
LD P_On
AND B_SYS_manual  ; 系统手动（总）
AND HMI_B_ZKXP2  ; 下料真空电磁阀
LD PLC11_103_step  ; PLC11步103
OR PLC11_116_step  ; PLC11步116
OR PLC11_126_step  ; PLC11步126
OR PLC11_136_step  ; PLC11步136
OR PLC11_146_step  ; PLC11步146
ORLD
OUT Q_B_ZKXP2  ; 下料真空电磁阀
TIM 210 #600  ; 下料真空电磁阀
; rung 10
LD P_On
AND B_SYS_manual  ; 系统手动（总）
AND HMI_B_CQF  ; 吹气电磁阀
OUT Q_B_CQF  ; 吹气电磁阀
TIM 211 #600  ; 吹气电磁阀
; rung 11
LD P_On
AND B_SYS_manual  ; 系统手动（总）
AND HMI_B_BJ1_QD  ; 步进1启动
OR PLC11_033_step  ; PLC11步033
OR PLC11_044_step  ; PLC11步044
OUT Q_B_BJ1_QD  ; 步进1启动

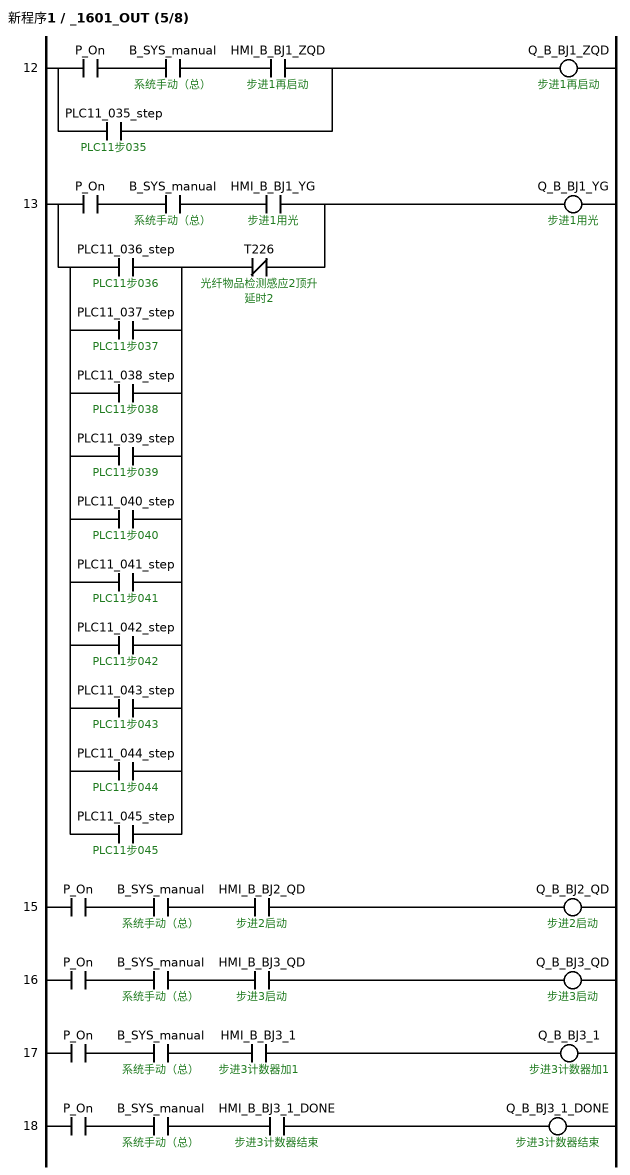
; rung 12
LD P_On
AND B_SYS_manual  ; 系统手动（总）
AND HMI_B_BJ1_ZQD  ; 步进1再启动
OR PLC11_035_step  ; PLC11步035
OUT Q_B_BJ1_ZQD  ; 步进1再启动
; rung 13
LD P_On
AND B_SYS_manual  ; 系统手动（总）
AND HMI_B_BJ1_YG  ; 步进1用光
LD PLC11_036_step  ; PLC11步036
OR PLC11_037_step  ; PLC11步037
OR PLC11_038_step  ; PLC11步038
OR PLC11_039_step  ; PLC11步039
OR PLC11_040_step  ; PLC11步040
OR PLC11_041_step  ; PLC11步041
OR PLC11_042_step  ; PLC11步042
OR PLC11_043_step  ; PLC11步043
OR PLC11_044_step  ; PLC11步044
OR PLC11_045_step  ; PLC11步045
ANDNOT T226  ; 光纤物品检测感应2顶升延时2
ORLD
OUT Q_B_BJ1_YG  ; 步进1用光
; rung 15
LD P_On
AND B_SYS_manual  ; 系统手动（总）
AND HMI_B_BJ2_QD  ; 步进2启动
OUT Q_B_BJ2_QD  ; 步进2启动
; rung 16
LD P_On
AND B_SYS_manual  ; 系统手动（总）
AND HMI_B_BJ3_QD  ; 步进3启动
OUT Q_B_BJ3_QD  ; 步进3启动
; rung 17
LD P_On
AND B_SYS_manual  ; 系统手动（总）
AND HMI_B_BJ3_1  ; 步进3计数器加1
OUT Q_B_BJ3_1  ; 步进3计数器加1
; rung 18
LD P_On
AND B_SYS_manual  ; 系统手动（总）
AND HMI_B_BJ3_1_DONE  ; 步进3计数器结束
OUT Q_B_BJ3_1_DONE  ; 步进3计数器结束

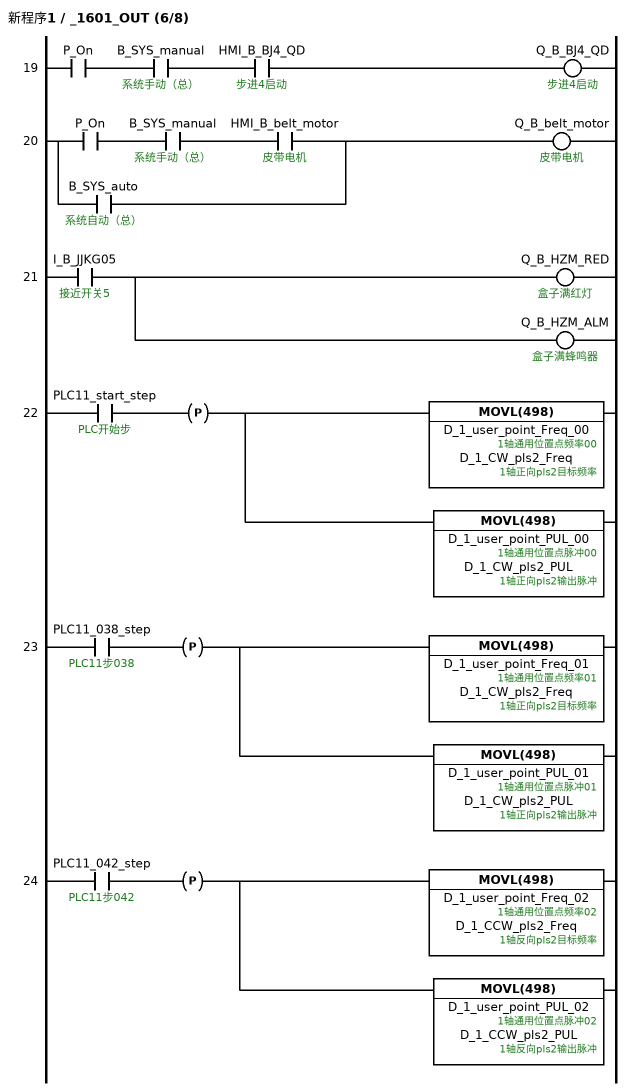
; rung 19
LD P_On
AND B_SYS_manual  ; 系统手动（总）
AND HMI_B_BJ4_QD  ; 步进4启动
OUT Q_B_BJ4_QD  ; 步进4启动
; rung 20
LD P_On
AND B_SYS_manual  ; 系统手动（总）
AND HMI_B_belt_motor  ; 皮带电机
OR B_SYS_auto  ; 系统自动（总）
OUT Q_B_belt_motor  ; 皮带电机
; rung 21
LD I_B_JJKG05  ; 接近开关5
OUT Q_B_HZM_RED  ; 盒子满红灯
OUT Q_B_HZM_ALM  ; 盒子满蜂鸣器
; rung 22
LD PLC11_start_step  ; PLC开始步
UP(521)
MOVL(498) D_1_user_point_Freq_00 D_1_CW_pls2_Freq  ; 1轴通用位置点频率00, 1轴正向pls2目标频率
MOVL(498) D_1_user_point_PUL_00 D_1_CW_pls2_PUL  ; 1轴通用位置点脉冲00, 1轴正向pls2输出脉冲
; rung 23
LD PLC11_038_step  ; PLC11步038
UP(521)
MOVL(498) D_1_user_point_Freq_01 D_1_CW_pls2_Freq  ; 1轴通用位置点频率01, 1轴正向pls2目标频率
MOVL(498) D_1_user_point_PUL_01 D_1_CW_pls2_PUL  ; 1轴通用位置点脉冲01, 1轴正向pls2输出脉冲
; rung 24
LD PLC11_042_step  ; PLC11步042
UP(521)
MOVL(498) D_1_user_point_Freq_02 D_1_CCW_pls2_Freq  ; 1轴通用位置点频率02, 1轴反向pls2目标频率
MOVL(498) D_1_user_point_PUL_02 D_1_CCW_pls2_PUL  ; 1轴通用位置点脉冲02, 1轴反向pls2输出脉冲

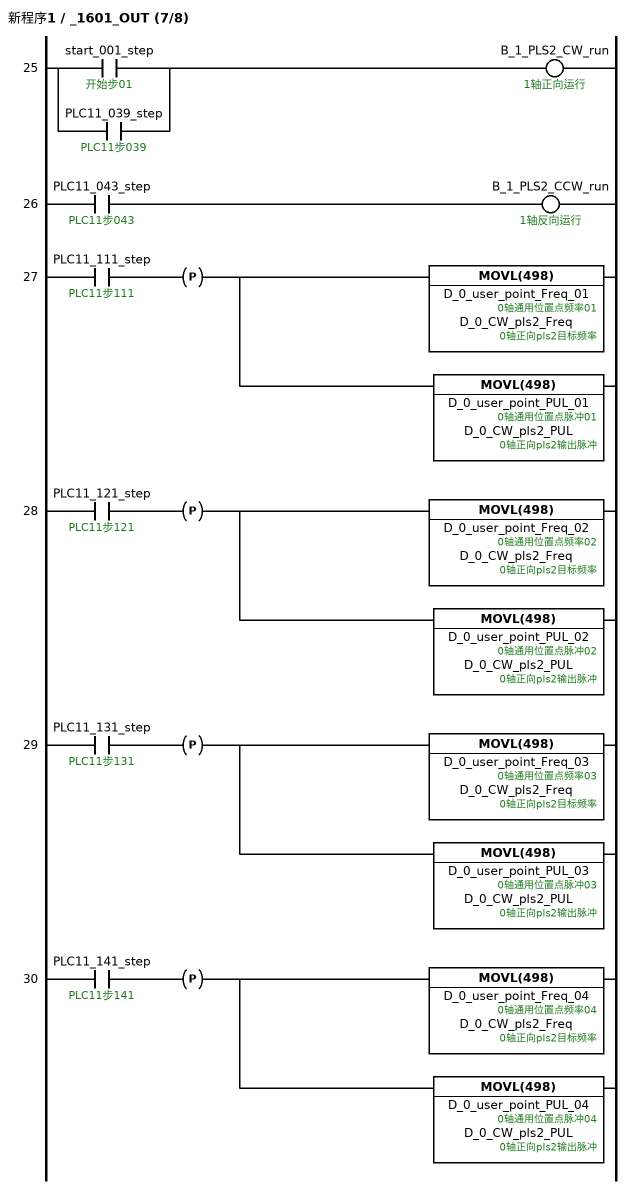
; rung 25
LD start_001_step  ; 开始步01
OR PLC11_039_step  ; PLC11步039
OUT B_1_PLS2_CW_run  ; 1轴正向运行
; rung 26
LD PLC11_043_step  ; PLC11步043
OUT B_1_PLS2_CCW_run  ; 1轴反向运行
; rung 27
LD PLC11_111_step  ; PLC11步111
UP(521)
MOVL(498) D_0_user_point_Freq_01 D_0_CW_pls2_Freq  ; 0轴通用位置点频率01, 0轴正向pls2目标频率
MOVL(498) D_0_user_point_PUL_01 D_0_CW_pls2_PUL  ; 0轴通用位置点脉冲01, 0轴正向pls2输出脉冲
; rung 28
LD PLC11_121_step  ; PLC11步121
UP(521)
MOVL(498) D_0_user_point_Freq_02 D_0_CW_pls2_Freq  ; 0轴通用位置点频率02, 0轴正向pls2目标频率
MOVL(498) D_0_user_point_PUL_02 D_0_CW_pls2_PUL  ; 0轴通用位置点脉冲02, 0轴正向pls2输出脉冲
; rung 29
LD PLC11_131_step  ; PLC11步131
UP(521)
MOVL(498) D_0_user_point_Freq_03 D_0_CW_pls2_Freq  ; 0轴通用位置点频率03, 0轴正向pls2目标频率
MOVL(498) D_0_user_point_PUL_03 D_0_CW_pls2_PUL  ; 0轴通用位置点脉冲03, 0轴正向pls2输出脉冲
; rung 30
LD PLC11_141_step  ; PLC11步141
UP(521)
MOVL(498) D_0_user_point_Freq_04 D_0_CW_pls2_Freq  ; 0轴通用位置点频率04, 0轴正向pls2目标频率
MOVL(498) D_0_user_point_PUL_04 D_0_CW_pls2_PUL  ; 0轴通用位置点脉冲04, 0轴正向pls2输出脉冲

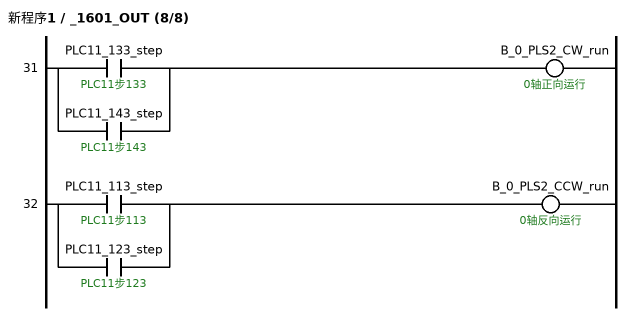
; rung 31
LD PLC11_133_step  ; PLC11步133
OR PLC11_143_step  ; PLC11步143
OUT B_0_PLS2_CW_run  ; 0轴正向运行
; rung 32
LD PLC11_113_step  ; PLC11步113
OR PLC11_123_step  ; PLC11步123
OUT B_0_PLS2_CCW_run  ; 0轴反向运行

### Section _1601_AUTO_INIT

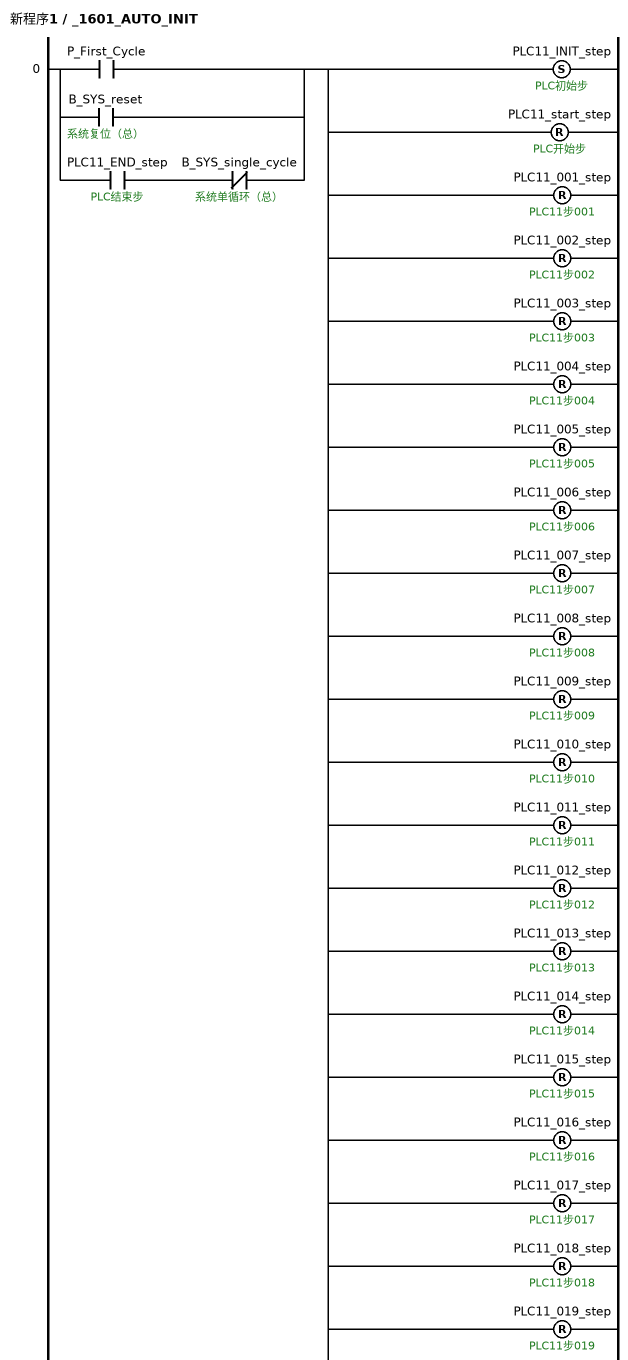

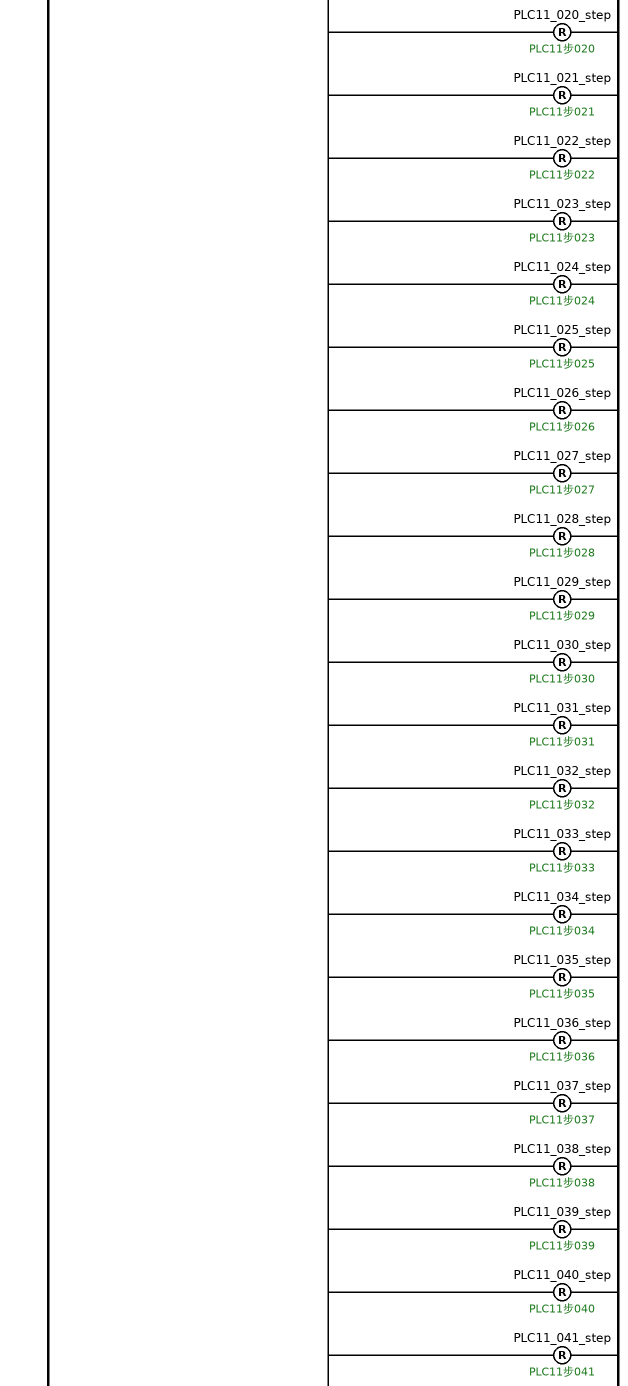

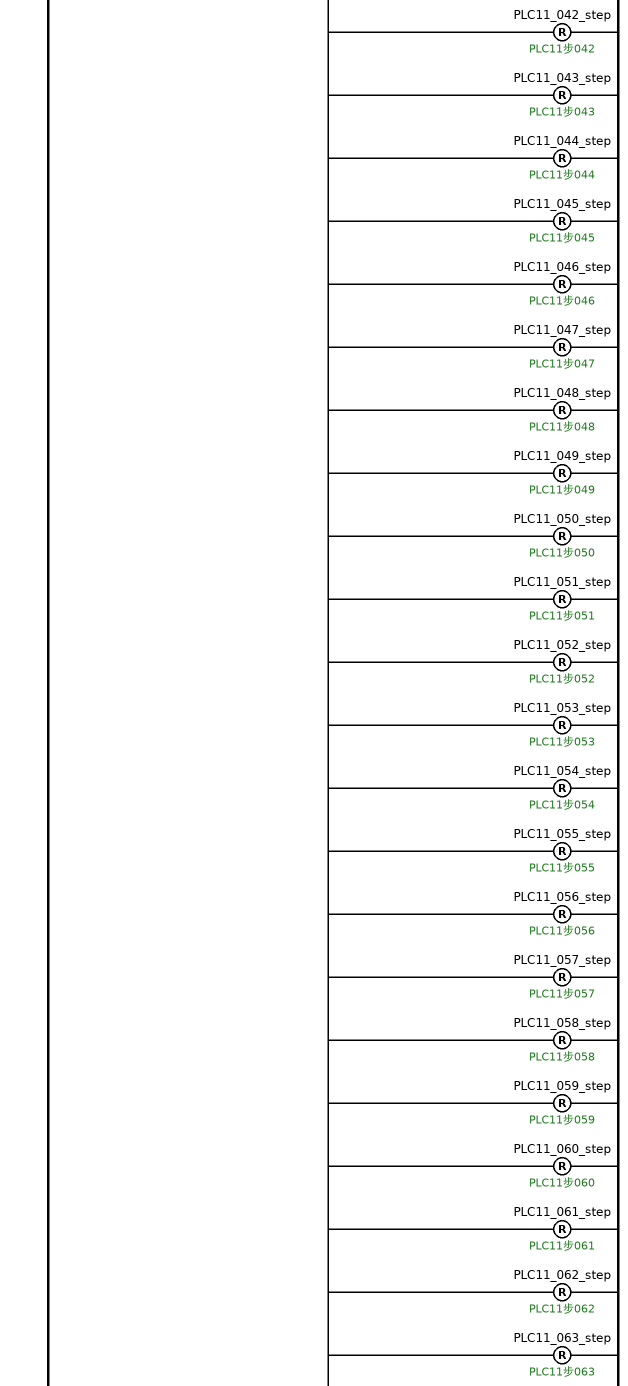

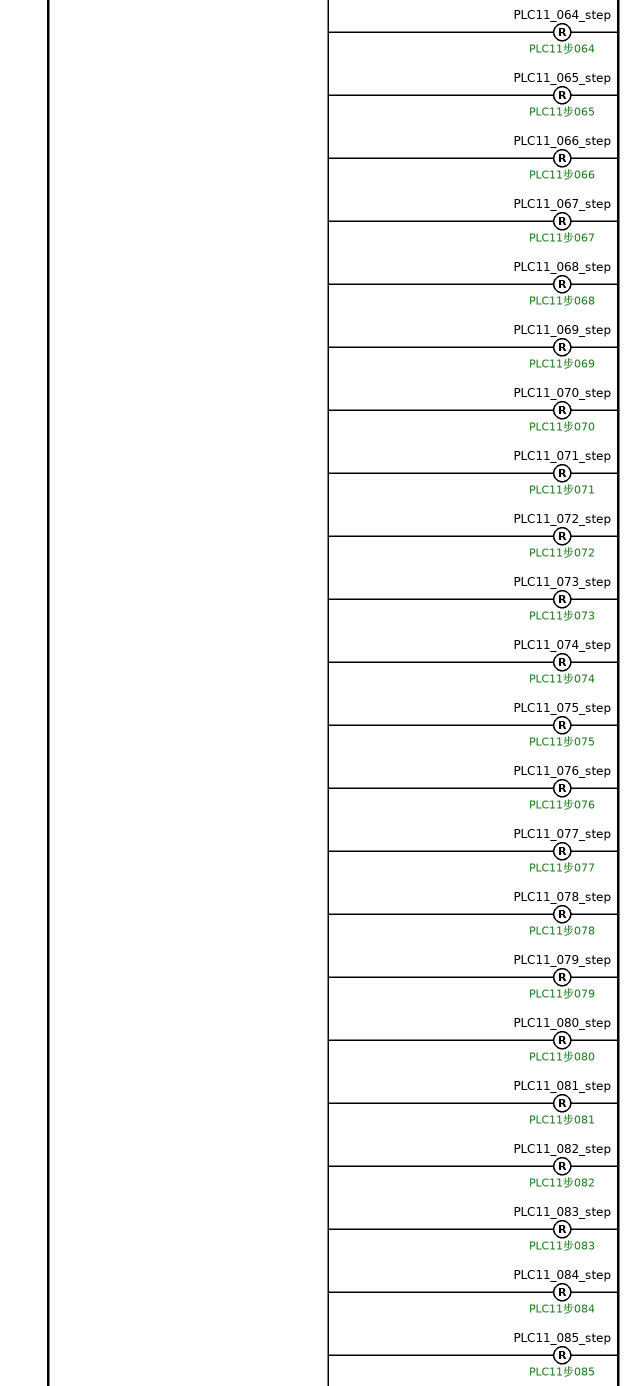

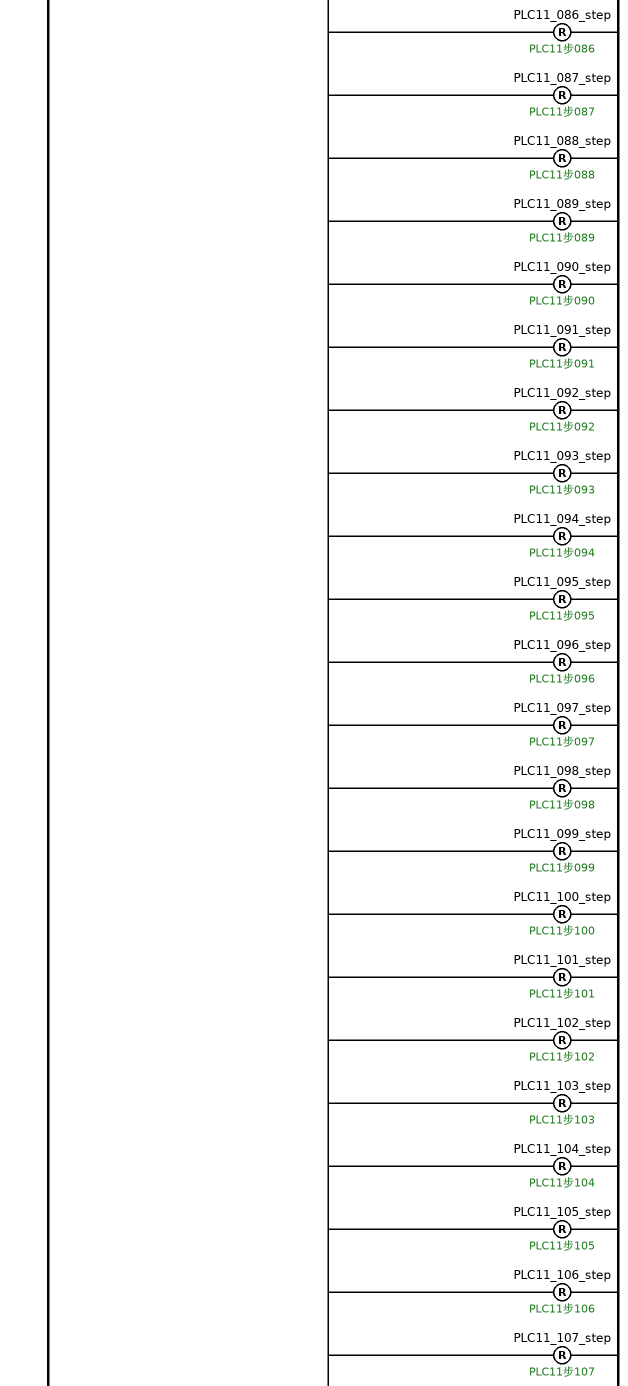

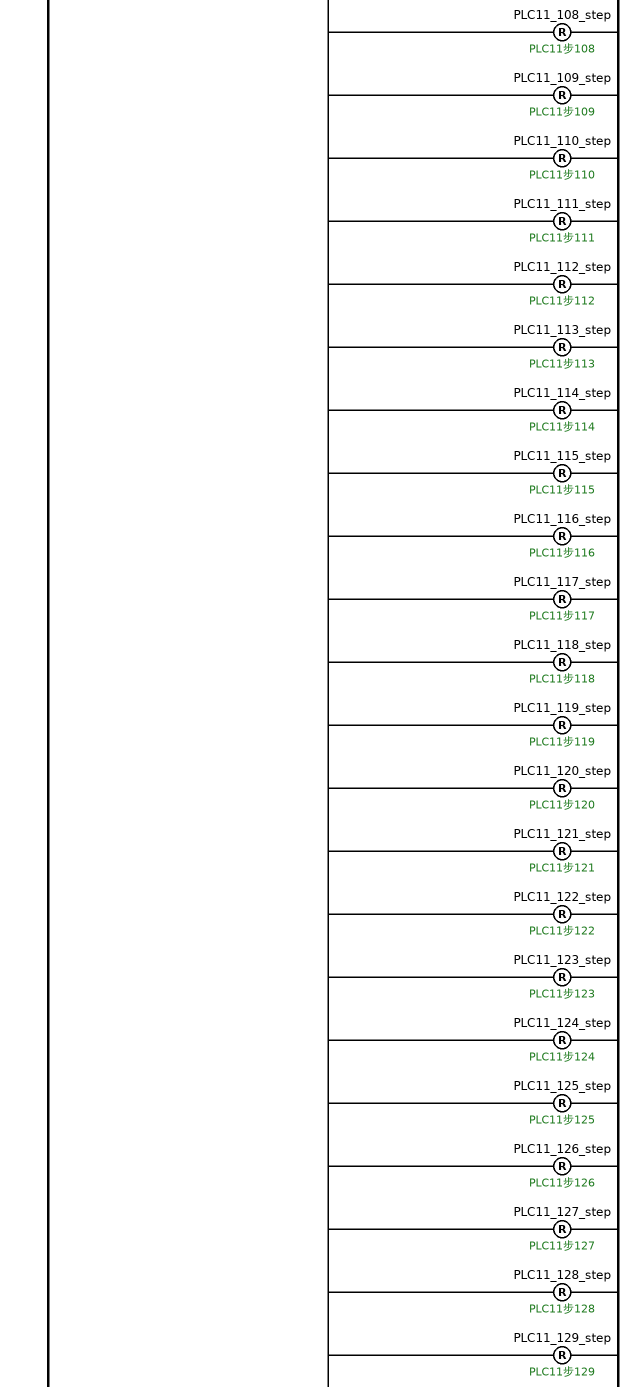

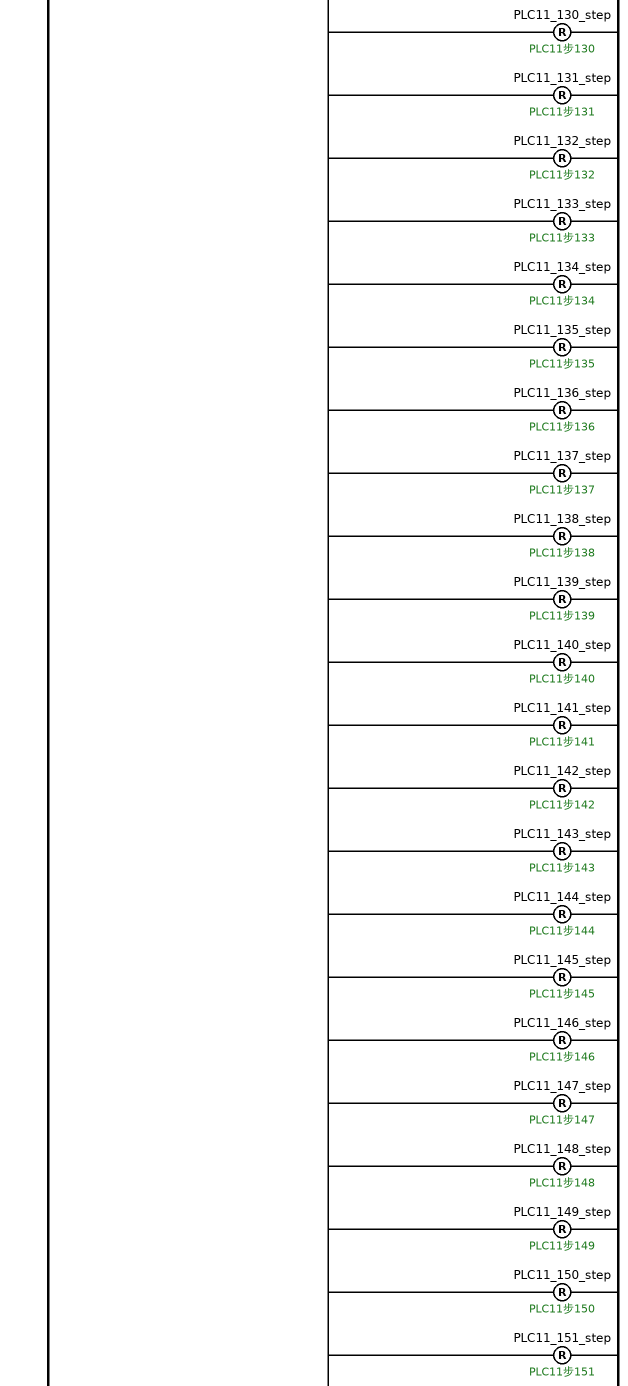

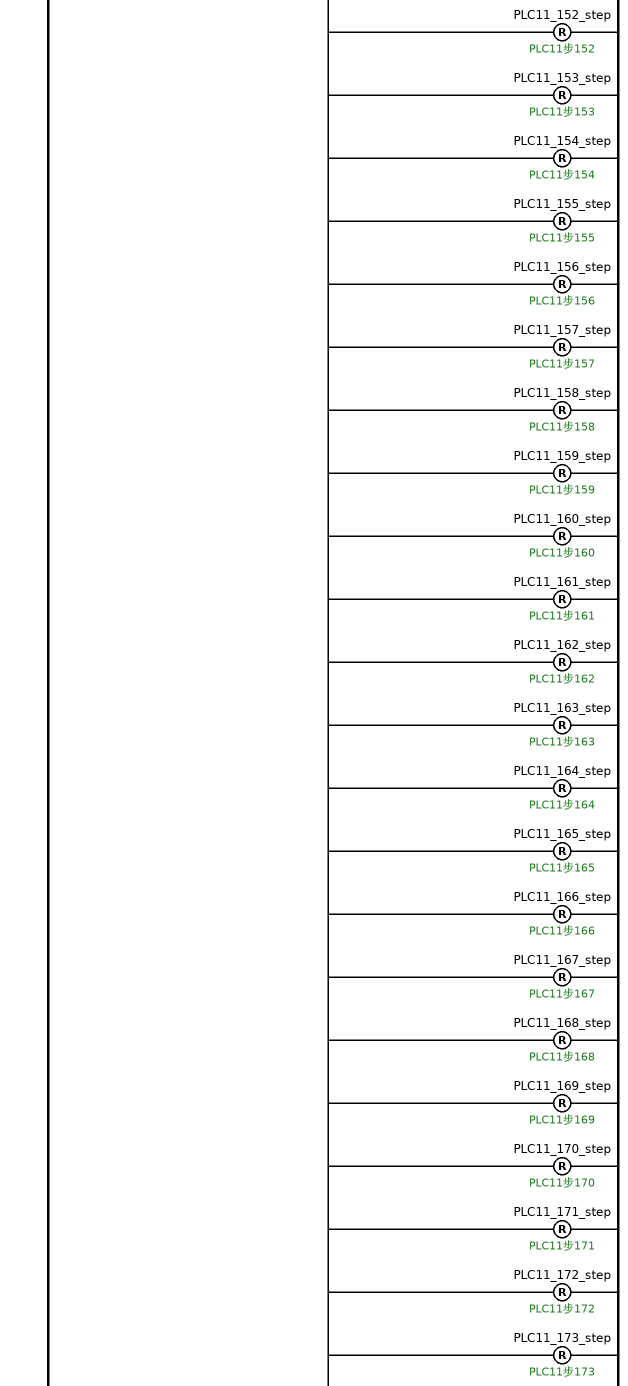

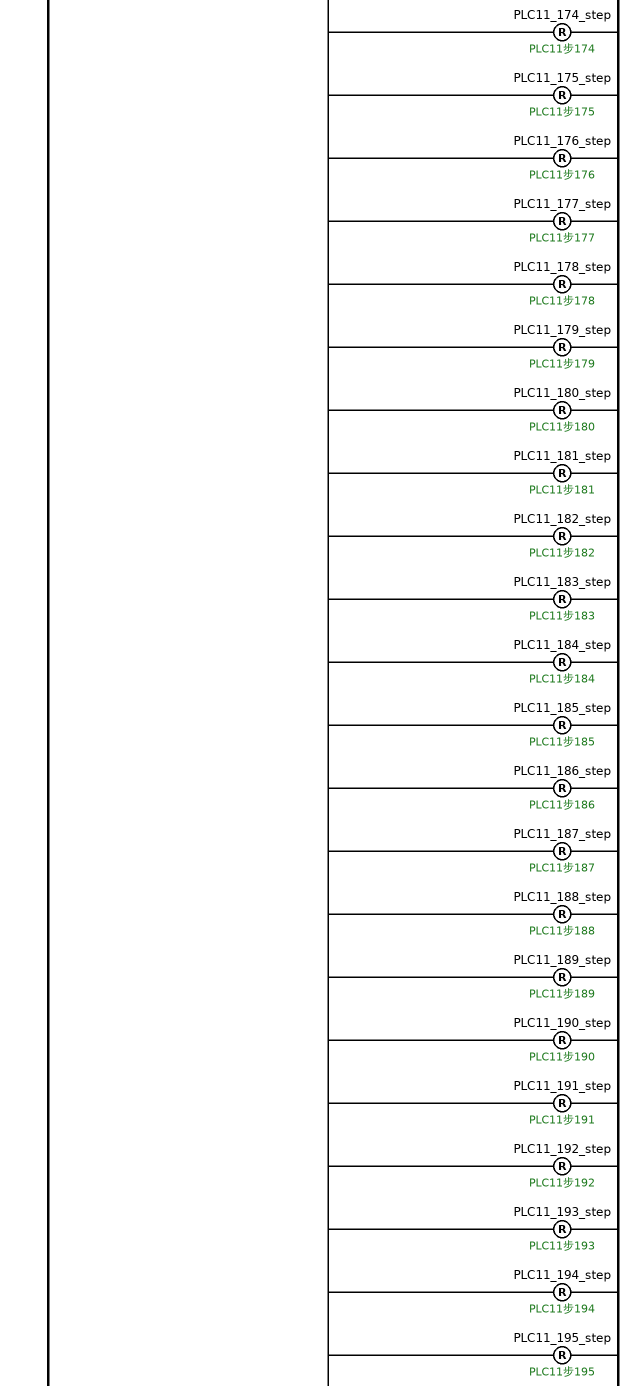

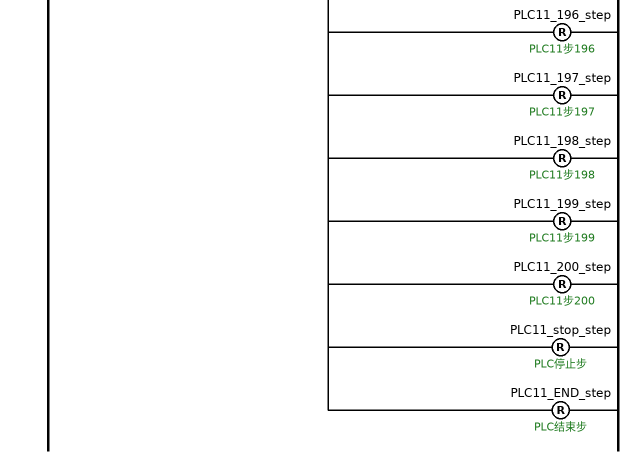
; rung 0
LD P_First_Cycle
OR B_SYS_reset  ; 系统复位（总）
LD PLC11_END_step  ; PLC结束步
ANDNOT B_SYS_single_cycle  ; 系统单循环（总）
ORLD
SET PLC11_INIT_step  ; PLC初始步
RSET PLC11_start_step  ; PLC开始步
RSET PLC11_001_step  ; PLC11步001
RSET PLC11_002_step  ; PLC11步002
RSET PLC11_003_step  ; PLC11步003
RSET PLC11_004_step  ; PLC11步004
RSET PLC11_005_step  ; PLC11步005
RSET PLC11_006_step  ; PLC11步006
RSET PLC11_007_step  ; PLC11步007
RSET PLC11_008_step  ; PLC11步008
RSET PLC11_009_step  ; PLC11步009
RSET PLC11_010_step  ; PLC11步010
RSET PLC11_011_step  ; PLC11步011
RSET PLC11_012_step  ; PLC11步012
RSET PLC11_013_step  ; PLC11步013
RSET PLC11_014_step  ; PLC11步014
RSET PLC11_015_step  ; PLC11步015
RSET PLC11_016_step  ; PLC11步016
RSET PLC11_017_step  ; PLC11步017
RSET PLC11_018_step  ; PLC11步018
RSET PLC11_019_step  ; PLC11步019
RSET PLC11_020_step  ; PLC11步020
RSET PLC11_021_step  ; PLC11步021
RSET PLC11_022_step  ; PLC11步022
RSET PLC11_023_step  ; PLC11步023
RSET PLC11_024_step  ; PLC11步024
RSET PLC11_025_step  ; PLC11步025
RSET PLC11_026_step  ; PLC11步026
RSET PLC11_027_step  ; PLC11步027
RSET PLC11_028_step  ; PLC11步028
RSET PLC11_029_step  ; PLC11步029
RSET PLC11_030_step  ; PLC11步030
RSET PLC11_031_step  ; PLC11步031
RSET PLC11_032_step  ; PLC11步032
RSET PLC11_033_step  ; PLC11步033
RSET PLC11_034_step  ; PLC11步034
RSET PLC11_035_step  ; PLC11步035
RSET PLC11_036_step  ; PLC11步036
RSET PLC11_037_step  ; PLC11步037
RSET PLC11_038_step  ; PLC11步038
RSET PLC11_039_step  ; PLC11步039
RSET PLC11_040_step  ; PLC11步040
RSET PLC11_041_step  ; PLC11步041
RSET PLC11_042_step  ; PLC11步042
RSET PLC11_043_step  ; PLC11步043
RSET PLC11_044_step  ; PLC11步044
RSET PLC11_045_step  ; PLC11步045
RSET PLC11_046_step  ; PLC11步046
RSET PLC11_047_step  ; PLC11步047
RSET PLC11_048_step  ; PLC11步048
RSET PLC11_049_step  ; PLC11步049
RSET PLC11_050_step  ; PLC11步050
RSET PLC11_051_step  ; PLC11步051
RSET PLC11_052_step  ; PLC11步052
RSET PLC11_053_step  ; PLC11步053
RSET PLC11_054_step  ; PLC11步054
RSET PLC11_055_step  ; PLC11步055
RSET PLC11_056_step  ; PLC11步056
RSET PLC11_057_step  ; PLC11步057
RSET PLC11_058_step  ; PLC11步058
RSET PLC11_059_step  ; PLC11步059
RSET PLC11_060_step  ; PLC11步060
RSET PLC11_061_step  ; PLC11步061
RSET PLC11_062_step  ; PLC11步062
RSET PLC11_063_step  ; PLC11步063
RSET PLC11_064_step  ; PLC11步064
RSET PLC11_065_step  ; PLC11步065
RSET PLC11_066_step  ; PLC11步066
RSET PLC11_067_step  ; PLC11步067
RSET PLC11_068_step  ; PLC11步068
RSET PLC11_069_step  ; PLC11步069
RSET PLC11_070_step  ; PLC11步070
RSET PLC11_071_step  ; PLC11步071
RSET PLC11_072_step  ; PLC11步072
RSET PLC11_073_step  ; PLC11步073
RSET PLC11_074_step  ; PLC11步074
RSET PLC11_075_step  ; PLC11步075
RSET PLC11_076_step  ; PLC11步076
RSET PLC11_077_step  ; PLC11步077
RSET PLC11_078_step  ; PLC11步078
RSET PLC11_079_step  ; PLC11步079
RSET PLC11_080_step  ; PLC11步080
RSET PLC11_081_step  ; PLC11步081
RSET PLC11_082_step  ; PLC11步082
RSET PLC11_083_step  ; PLC11步083
RSET PLC11_084_step  ; PLC11步084
RSET PLC11_085_step  ; PLC11步085
RSET PLC11_086_step  ; PLC11步086
RSET PLC11_087_step  ; PLC11步087
RSET PLC11_088_step  ; PLC11步088
RSET PLC11_089_step  ; PLC11步089
RSET PLC11_090_step  ; PLC11步090
RSET PLC11_091_step  ; PLC11步091
RSET PLC11_092_step  ; PLC11步092
RSET PLC11_093_step  ; PLC11步093
RSET PLC11_094_step  ; PLC11步094
RSET PLC11_095_step  ; PLC11步095
RSET PLC11_096_step  ; PLC11步096
RSET PLC11_097_step  ; PLC11步097
RSET PLC11_098_step  ; PLC11步098
RSET PLC11_099_step  ; PLC11步099
RSET PLC11_100_step  ; PLC11步100
RSET PLC11_101_step  ; PLC11步101
RSET PLC11_102_step  ; PLC11步102
RSET PLC11_103_step  ; PLC11步103
RSET PLC11_104_step  ; PLC11步104
RSET PLC11_105_step  ; PLC11步105
RSET PLC11_106_step  ; PLC11步106
RSET PLC11_107_step  ; PLC11步107
RSET PLC11_108_step  ; PLC11步108
RSET PLC11_109_step  ; PLC11步109
RSET PLC11_110_step  ; PLC11步110
RSET PLC11_111_step  ; PLC11步111
RSET PLC11_112_step  ; PLC11步112
RSET PLC11_113_step  ; PLC11步113
RSET PLC11_114_step  ; PLC11步114
RSET PLC11_115_step  ; PLC11步115
RSET PLC11_116_step  ; PLC11步116
RSET PLC11_117_step  ; PLC11步117
RSET PLC11_118_step  ; PLC11步118
RSET PLC11_119_step  ; PLC11步119
RSET PLC11_120_step  ; PLC11步120
RSET PLC11_121_step  ; PLC11步121
RSET PLC11_122_step  ; PLC11步122
RSET PLC11_123_step  ; PLC11步123
RSET PLC11_124_step  ; PLC11步124
RSET PLC11_125_step  ; PLC11步125
RSET PLC11_126_step  ; PLC11步126
RSET PLC11_127_step  ; PLC11步127
RSET PLC11_128_step  ; PLC11步128
RSET PLC11_129_step  ; PLC11步129
RSET PLC11_130_step  ; PLC11步130
RSET PLC11_131_step  ; PLC11步131
RSET PLC11_132_step  ; PLC11步132
RSET PLC11_133_step  ; PLC11步133
RSET PLC11_134_step  ; PLC11步134
RSET PLC11_135_step  ; PLC11步135
RSET PLC11_136_step  ; PLC11步136
RSET PLC11_137_step  ; PLC11步137
RSET PLC11_138_step  ; PLC11步138
RSET PLC11_139_step  ; PLC11步139
RSET PLC11_140_step  ; PLC11步140
RSET PLC11_141_step  ; PLC11步141
RSET PLC11_142_step  ; PLC11步142
RSET PLC11_143_step  ; PLC11步143
RSET PLC11_144_step  ; PLC11步144
RSET PLC11_145_step  ; PLC11步145
RSET PLC11_146_step  ; PLC11步146
RSET PLC11_147_step  ; PLC11步147
RSET PLC11_148_step  ; PLC11步148
RSET PLC11_149_step  ; PLC11步149
RSET PLC11_150_step  ; PLC11步150
RSET PLC11_151_step  ; PLC11步151
RSET PLC11_152_step  ; PLC11步152
RSET PLC11_153_step  ; PLC11步153
RSET PLC11_154_step  ; PLC11步154
RSET PLC11_155_step  ; PLC11步155
RSET PLC11_156_step  ; PLC11步156
RSET PLC11_157_step  ; PLC11步157
RSET PLC11_158_step  ; PLC11步158
RSET PLC11_159_step  ; PLC11步159
RSET PLC11_160_step  ; PLC11步160
RSET PLC11_161_step  ; PLC11步161
RSET PLC11_162_step  ; PLC11步162
RSET PLC11_163_step  ; PLC11步163
RSET PLC11_164_step  ; PLC11步164
RSET PLC11_165_step  ; PLC11步165
RSET PLC11_166_step  ; PLC11步166
RSET PLC11_167_step  ; PLC11步167
RSET PLC11_168_step  ; PLC11步168
RSET PLC11_169_step  ; PLC11步169
RSET PLC11_170_step  ; PLC11步170
RSET PLC11_171_step  ; PLC11步171
RSET PLC11_172_step  ; PLC11步172
RSET PLC11_173_step  ; PLC11步173
RSET PLC11_174_step  ; PLC11步174
RSET PLC11_175_step  ; PLC11步175
RSET PLC11_176_step  ; PLC11步176
RSET PLC11_177_step  ; PLC11步177
RSET PLC11_178_step  ; PLC11步178
RSET PLC11_179_step  ; PLC11步179
RSET PLC11_180_step  ; PLC11步180
RSET PLC11_181_step  ; PLC11步181
RSET PLC11_182_step  ; PLC11步182
RSET PLC11_183_step  ; PLC11步183
RSET PLC11_184_step  ; PLC11步184
RSET PLC11_185_step  ; PLC11步185
RSET PLC11_186_step  ; PLC11步186
RSET PLC11_187_step  ; PLC11步187
RSET PLC11_188_step  ; PLC11步188
RSET PLC11_189_step  ; PLC11步189
RSET PLC11_190_step  ; PLC11步190
RSET PLC11_191_step  ; PLC11步191
RSET PLC11_192_step  ; PLC11步192
RSET PLC11_193_step  ; PLC11步193
RSET PLC11_194_step  ; PLC11步194
RSET PLC11_195_step  ; PLC11步195
RSET PLC11_196_step  ; PLC11步196
RSET PLC11_197_step  ; PLC11步197
RSET PLC11_198_step  ; PLC11步198
RSET PLC11_199_step  ; PLC11步199
RSET PLC11_200_step  ; PLC11步200
RSET PLC11_stop_step  ; PLC停止步
RSET PLC11_END_step  ; PLC结束步

### Section _1601_AUTO_1

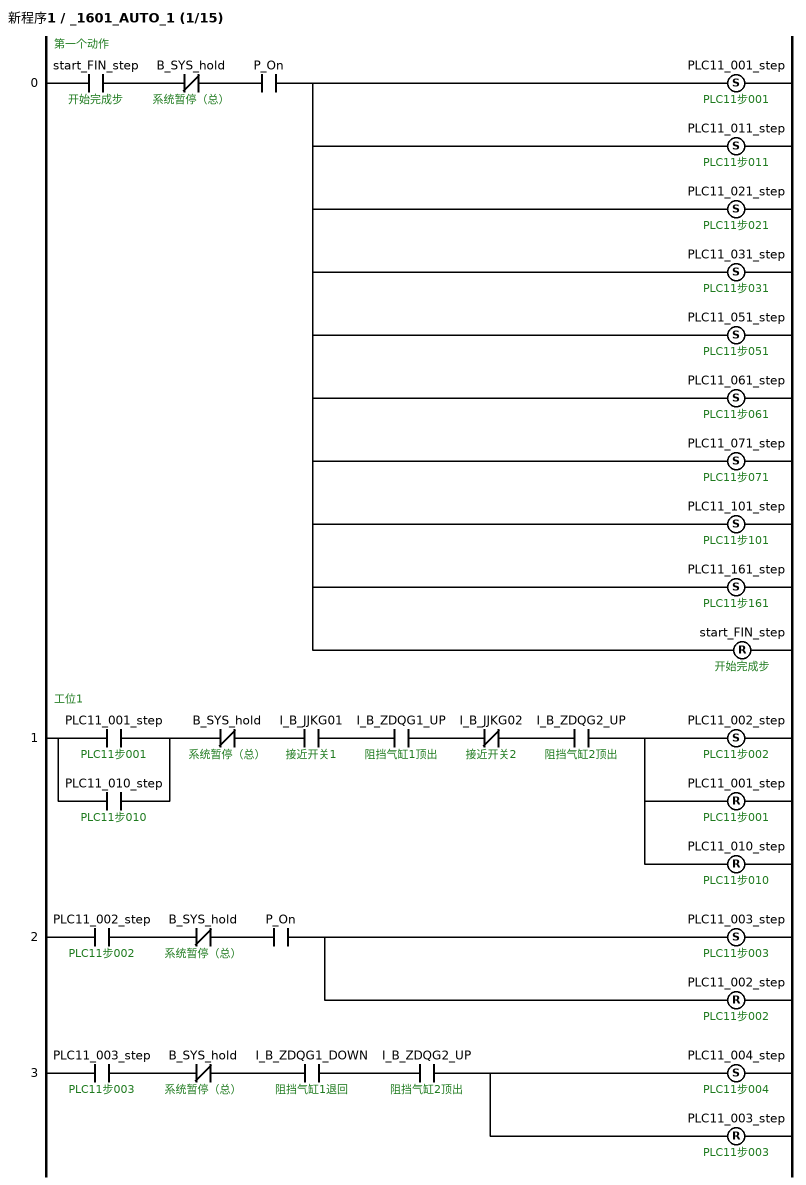
; rung 0: 第一个动作
LD start_FIN_step  ; 开始完成步
ANDNOT B_SYS_hold  ; 系统暂停（总）
AND P_On
SET PLC11_001_step  ; PLC11步001
SET PLC11_011_step  ; PLC11步011
SET PLC11_021_step  ; PLC11步021
SET PLC11_031_step  ; PLC11步031
SET PLC11_051_step  ; PLC11步051
SET PLC11_061_step  ; PLC11步061
SET PLC11_071_step  ; PLC11步071
SET PLC11_101_step  ; PLC11步101
SET PLC11_161_step  ; PLC11步161
RSET start_FIN_step  ; 开始完成步
; rung 1: 工位1
LD PLC11_001_step  ; PLC11步001
OR PLC11_010_step  ; PLC11步010
ANDNOT B_SYS_hold  ; 系统暂停（总）
AND I_B_JJKG01  ; 接近开关1
AND I_B_ZDQG1_UP  ; 阻挡气缸1顶出
ANDNOT I_B_JJKG02  ; 接近开关2
AND I_B_ZDQG2_UP  ; 阻挡气缸2顶出
SET PLC11_002_step  ; PLC11步002
RSET PLC11_001_step  ; PLC11步001
RSET PLC11_010_step  ; PLC11步010
; rung 2
LD PLC11_002_step  ; PLC11步002
ANDNOT B_SYS_hold  ; 系统暂停（总）
AND P_On
SET PLC11_003_step  ; PLC11步003
RSET PLC11_002_step  ; PLC11步002
; rung 3
LD PLC11_003_step  ; PLC11步003
ANDNOT B_SYS_hold  ; 系统暂停（总）
AND I_B_ZDQG1_DOWN  ; 阻挡气缸1退回
AND I_B_ZDQG2_UP  ; 阻挡气缸2顶出
SET PLC11_004_step  ; PLC11步004
RSET PLC11_003_step  ; PLC11步003

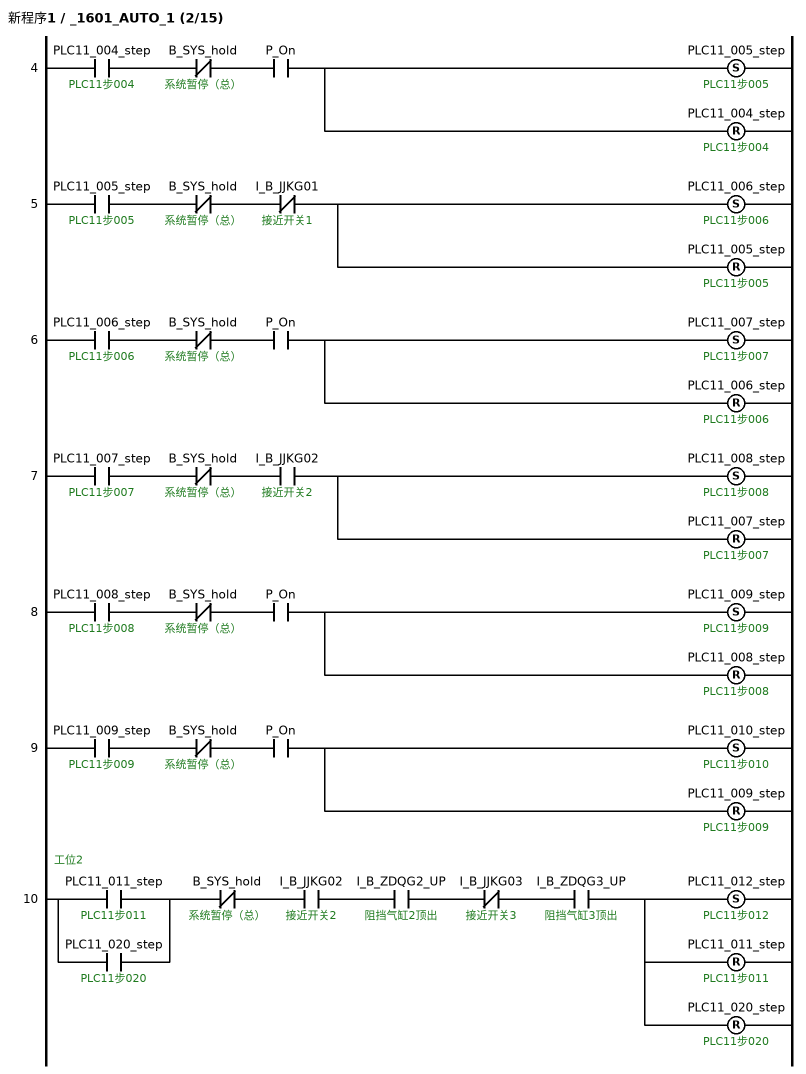
; rung 4
LD PLC11_004_step  ; PLC11步004
ANDNOT B_SYS_hold  ; 系统暂停（总）
AND P_On
SET PLC11_005_step  ; PLC11步005
RSET PLC11_004_step  ; PLC11步004
; rung 5
LD PLC11_005_step  ; PLC11步005
ANDNOT B_SYS_hold  ; 系统暂停（总）
ANDNOT I_B_JJKG01  ; 接近开关1
SET PLC11_006_step  ; PLC11步006
RSET PLC11_005_step  ; PLC11步005
; rung 6
LD PLC11_006_step  ; PLC11步006
ANDNOT B_SYS_hold  ; 系统暂停（总）
AND P_On
SET PLC11_007_step  ; PLC11步007
RSET PLC11_006_step  ; PLC11步006
; rung 7
LD PLC11_007_step  ; PLC11步007
ANDNOT B_SYS_hold  ; 系统暂停（总）
AND I_B_JJKG02  ; 接近开关2
SET PLC11_008_step  ; PLC11步008
RSET PLC11_007_step  ; PLC11步007
; rung 8
LD PLC11_008_step  ; PLC11步008
ANDNOT B_SYS_hold  ; 系统暂停（总）
AND P_On
SET PLC11_009_step  ; PLC11步009
RSET PLC11_008_step  ; PLC11步008
; rung 9
LD PLC11_009_step  ; PLC11步009
ANDNOT B_SYS_hold  ; 系统暂停（总）
AND P_On
SET PLC11_010_step  ; PLC11步010
RSET PLC11_009_step  ; PLC11步009
; rung 10: 工位2
LD PLC11_011_step  ; PLC11步011
OR PLC11_020_step  ; PLC11步020
ANDNOT B_SYS_hold  ; 系统暂停（总）
AND I_B_JJKG02  ; 接近开关2
AND I_B_ZDQG2_UP  ; 阻挡气缸2顶出
ANDNOT I_B_JJKG03  ; 接近开关3
AND I_B_ZDQG3_UP  ; 阻挡气缸3顶出
SET PLC11_012_step  ; PLC11步012
RSET PLC11_011_step  ; PLC11步011
RSET PLC11_020_step  ; PLC11步020

